fb_axis110_04Z(enIN_State       := enIN_State,
               parIN_Buttons    := ADR(AXIS.btTeachArAxis[Axis_e.ST110_04Z]),
               xIN_DisButtons   :=,
               xIN_Quit         := xIN_Quit,
               xIN_AX5000       := TRUE,
               xIN_ENC_ABS      := TRUE,
               xIN_PARAMok      := TRUE,
               xIN_FREE         := TRUE,
               xIN_FREE_HOME    := TRUE,
               rIN_POSMIN       := ST110_Axis.const110_04Z.POS_MIN,
               rIN_POSMAX       := ST110_Axis.const110_04Z.POS_MAX,
               rIN_VELOMAX      := ST110_Axis.const110_04Z.VELO_MAX,
               rIN_VELOMANU     := ST110_Axis.const110_04Z.VELO_MANU,
               rIN_VELOOPEN     := ST110_Axis.const110_04Z.VELO_MANU / 4,
               rIN_JogInc       := AXIS.rTeachIncAxis,
               rIN_VeloJogManu  := TO_REAL(AXIS.rJogVelo_pc),
               xIN_HomeExe      :=,
               xIN_HomeCalib    := FALSE,
               xIN_Execute      := fb_PnpVerAxisU.xOUT_Execute,
               xIN_Relative     := FALSE,
               rIN_Position     := LREAL_TO_REAL(fb_PnpVerAxisU.OUT_MoveProfile.lrPosition),
               rIN_Velocity     := LREAL_TO_REAL(fb_PnpVerAxisU.OUT_MoveProfile.lrVelocity),
               rIN_Acceleration := LREAL_TO_REAL(fb_PnpVerAxisU.OUT_MoveProfile.lrAccel),
               rIN_Deceleration := LREAL_TO_REAL(fb_PnpVerAxisU.OUT_MoveProfile.lrDecel),
               rIN_Jerk         := LREAL_TO_REAL(fb_PnpVerAxisU.OUT_MoveProfile.lrJerk),
               rIN_PosManu      :=
               TO_REAL(_20_AUTO.recipe
                           .linearAxis[LinearAxis_e.ST110_04Z].movesList[AXIS.bTeachPos[Axis_e.ST110_04Z]].lrPosition),
               xIN_Reset   := xIN_Reset,
               rOUT_ActPos => ST110_Axis.axis110_04Z.rActPos,
               axisIN_REF  := fb_simu_axis110_04Z.pOUT_axisRef^);

// pneumatics

fb_gripperLeft(xIN_Reset    := xIN_Reset OR (ST110_Pnp_e.RESET = iOUT_Step),
               xIN_Quit     := xIN_Quit,
               xIN_Manu     := enState.StateMANU = enIN_State,
               pbtIN_Button := ADR(HMI.btManuCylinders[StationList_e.ST110][1]),
               xIN_GS       := simu_gripperLeft.xOUT_inGS,
               xIN_AS       := simu_gripperLeft.xOUT_inAS,
               xIN_FREE     := TRUE,
               xINtoGS      := (ST110_Pnp_e.Vacum_off = iOUT_Step) OR (ST110_Pnp_e.Init_stop_vacum = iOUT_Step),
               xINtoAS      := _20_AUTO.recipe.st110.xUseVerLeft AND (ST110_Pnp_e.Vacum_on = iOUT_Step),
               tIN_ErrAS    := DINT_TO_TIME(_20_AUTO.recipe.cylinder2Pos[StationList_e.ST110]
                                                [ST110_Cylinders_e.VakuumgreiferLinks].toAS_alarm_time),
               tIN_ErrGS := DINT_TO_TIME(_20_AUTO.recipe.cylinder2Pos[StationList_e.ST110]
                                             [ST110_Cylinders_e.VakuumgreiferLinks].toGS_alarm_time),
               tIN_WaitAS := DINT_TO_TIME(_20_AUTO.recipe.cylinder2Pos[StationList_e.ST110]
                                              [ST110_Cylinders_e.VakuumgreiferLinks].toAS_wait_time),
               tIN_WaitGS := DINT_TO_TIME(_20_AUTO.recipe.cylinder2Pos[StationList_e.ST110]
                                              [ST110_Cylinders_e.VakuumgreiferLinks].toGS_wait_time));

simu_gripperLeft(xIN_Enable := TRUE, // PNP_SIMULATION AND CONST.USE_SIMULATION,
                 xIN_inGS   := (IO_BOX.I5500_ST110_vakumkontrolle_links / TO_INT(16#FFFF / 100)) <=
                               _20_AUTO.recipe.st110.vakum_left_pc,
                 xIN_inAS := (IO_BOX.I5500_ST110_vakumkontrolle_links / TO_INT(16#FFFF / 100)) >
                             _20_AUTO.recipe.st110.vakum_left_pc,
                 xIN_valve := fb_gripperLeft.xOUT_VALVE,
                 tIN_GS_ms := 200,  //ms
                 tIN_AS_ms := 200); //ms

fb_gripperRight(xIN_Reset    := xIN_Reset OR (ST110_Pnp_e.RESET = iOUT_Step),
                xIN_Quit     := xIN_Quit,
                xIN_Manu     := enState.StateMANU = enIN_State,
                pbtIN_Button := ADR(HMI.btManuCylinders[StationList_e.ST110][2]),
                xIN_GS       := simu_gripperRight.xOUT_inGS,
                xIN_AS       := simu_gripperRight.xOUT_inAS,
                xIN_FREE     := TRUE,
                xINtoGS      := (ST110_Pnp_e.Vacum_off = iOUT_Step) OR (ST110_Pnp_e.Init_stop_vacum = iOUT_Step),
                xINtoAS      := _20_AUTO.recipe.st110.xUseVerRight AND (ST110_Pnp_e.Vacum_on = iOUT_Step),
                tIN_ErrAS    := DINT_TO_TIME(_20_AUTO.recipe.cylinder2Pos[StationList_e.ST110]
                                                 [ST110_Cylinders_e.VakuumgreiferRechts].toAS_alarm_time),
                tIN_ErrGS := DINT_TO_TIME(_20_AUTO.recipe.cylinder2Pos[StationList_e.ST110]
                                              [ST110_Cylinders_e.VakuumgreiferRechts].toGS_alarm_time),
                tIN_WaitAS := DINT_TO_TIME(_20_AUTO.recipe.cylinder2Pos[StationList_e.ST110]
                                               [ST110_Cylinders_e.VakuumgreiferRechts].toAS_wait_time),
                tIN_WaitGS := DINT_TO_TIME(_20_AUTO.recipe.cylinder2Pos[StationList_e.ST110]
                                               [ST110_Cylinders_e.VakuumgreiferRechts].toGS_wait_time));

simu_gripperRight(xIN_Enable := TRUE, // PNP_SIMULATION AND CONST.USE_SIMULATION,
                  xIN_inGS   := (IO_BOX.I5600_ST110_vakumkontrolle_rechts / TO_INT(16#FFFF / 100)) <=
                                _20_AUTO.recipe.st110.vakum_right_pc,
                  xIN_inAS := (IO_BOX.I5600_ST110_vakumkontrolle_rechts / TO_INT(16#FFFF / 100)) >
                              _20_AUTO.recipe.st110.vakum_right_pc,
                  xIN_valve := fb_gripperRight.xOUT_VALVE,
                  tIN_GS_ms := 200,  //ms
                  tIN_AS_ms := 200); //ms

// kraft sensor
fb_kraftLeft(lrIN_MaxLimit := LREAL#2.0);
fb_kraftRight(lrIN_MaxLimit := LREAL#2.0);

(*******************************************************************)
(* OUTPUTS *)
(*******************************************************************)
// Error Flag 
xOUT_ErrFlag := (bOUT_Error <> 0) OR (ST110_Pnp_e.ERROR = iOUT_Step);
// Baustein befindet sich im Ablauf 
xOUT_Busy := (iOUT_Step > ST110_Pnp_e.READY) AND (iOUT_Step < ST110_Pnp_e.DONE);
// Baustein hat den Ablauf beendet
xOUT_Done := (iOUT_Step = ST110_Pnp_e.DONE);
// Process ready
xOUT_Ready := (iOUT_Step = ST110_Pnp_e.READY) OR (iOUT_Step = ST110_Pnp_e.waitOnMover);
// Timeout FB 				 		
xOUT_Timeout := TON_Timeout.Q;
// Itialisierung fertig			
xOUT_InitDone := (iOUT_Step = ST110_Pnp_e.READY) OR (iOUT_Step = ST110_Pnp_e.waitOnMover);
// Aktueller Schritt			
iOUT_Step := iOUT_Step; //Im Ablauf gesetzt		
sOUT_Step := TO_STRING(iOUT_Step);
//Fehlernummer	 
bOUT_Error := bOUT_Error; //Im Ablauf/FB gesetzt	
(* Warte (alle Schritte wo auf FG oder Teile gewartet wird) *)
xOUT_Wait := (iOUT_Step = ST110_Pnp_e.DONE) OR
             (iOUT_Step = ST110_Pnp_e.READY) OR
             (iOUT_Step = ST110_Pnp_e.START) OR
             (iOUT_Step = ST110_Pnp_e.waitOnMover) OR
             (iOUT_Step = ST110_Pnp_e.SYNC_MOVER_LEAVE) OR
             (iOUT_Step = ST110_Pnp_e.PnP_WaitOnFeeder);

xOUT_MoverFree := iOUT_Step >= ST110_Pnp_e.MOVER_FREE_OP AND iOUT_Step < ST110_Pnp_e.MOVER_NEEDED_OP;

iOUT_ProcessCompletion := F_GetPercent_2(iOUT_Step,
                                         ST110_Pnp_e.PnP_Hor_ToRotTablePos,
                                         ST110_Pnp_e.PnP_Hor_ToTrackPos,
                                         ST110_Pnp_e.PnP_Ver_ShuttleDown,
                                         ST110_Pnp_e.PnP_Ver_ShuttleUp);

xOUT_PickPiece := iOUT_Step = ST110_Pnp_e.PnP_Hor_ToTrackPos;

OUT.Q104_ST110_vacum_on_left  := fb_gripperLeft.xOUT_VALVE AND NOT (PNP_SIMULATION AND CONST.USE_SIMULATION);
OUT.Q105_ST110_vacum_on_right := fb_gripperRight.xOUT_VALVE AND NOT (PNP_SIMULATION AND CONST.USE_SIMULATION);

IF NOT IN.I004_druckwachter_luftdruck_ok THEN
    xIsPiecesPicked := FALSE;
END_IF

(*******************************************************************)
(* Ablauf *)
(*******************************************************************)

(* Sperren *)
IF xIN_Sperre THEN
    iPreStep  := ST110_Pnp_e.RESET;
    iOUT_Step := ST110_Pnp_e.RESET;
    RETURN;
END_IF;

(* Schritt Merker *)
IF iAktStep <> iOUT_Step THEN
    iLastStep := iAktStep;
    iAktStep  := iOUT_Step;
END_IF

(* START *)
rtSTART(CLK := xIN_Start);

IF 0 = bOUT_Error THEN
    IF fb_axis110_01Y.xOUT_ErrFlag THEN
        bOUT_Error := ST110_Alarm_e.Axis_110_01Y_error;
    ELSIF fb_axis110_02Z.xOUT_ErrFlag THEN
        bOUT_Error := ST110_Alarm_e.Axis_110_02Z_error;
    ELSIF fb_axis110_03Z.xOUT_ErrFlag THEN
        bOUT_Error := ST110_Alarm_e.Axis_110_03Z_error;
    ELSIF fb_axis110_04Z.xOUT_ErrFlag THEN
        bOUT_Error := ST110_Alarm_e.Axis_110_04Z_error;
    ELSIF fb_gripperLeft.xOUT_ErrFlag THEN
        bOUT_Error := ST110_Alarm_e.Cylinder_vacuum_griper_left;
    ELSIF fb_gripperRight.xOUT_ErrFlag THEN
        bOUT_Error := ST110_Alarm_e.Cylinder_vacuum_griper_right;
    END_IF
ELSIF iOUT_Step < ST110_Pnp_e.ERROR THEN
    iPreStep  := ST110_Pnp_e.INIT;
    iOUT_Step := ST110_Pnp_e.ERROR;
END_IF

(*******************************************************************)
(* Schrittkette  *)
(*******************************************************************)
CASE iOUT_Step OF

(***** RESET *****)
ST110_Pnp_e.RESET: (* Schritt 0-99 *)
    //Initialisierungen
    //Start Init Ablauf
    IF xIN_Init THEN
        iOUT_Step := ST110_Pnp_e.INIT;
        //Start Manu Ablauf
    ELSIF enIN_State = StateMANU AND xIN_NextStep THEN
        iOUT_Step := ST110_Pnp_e.INIT;
    END_IF;

(***** INIT *****)
ST110_Pnp_e.INIT: (* Grundstellung ? *)
    iOUT_Step := ST110_Pnp_e.Init_VerticalUp_04;

ST110_Pnp_e.Init_VerticalUp_04:
    IF fb_PnpVerAxisU.MoveTo(ST110_PnpVerPushPos_e.down).xOUT_InPos THEN
        iOUT_Step := ST110_Pnp_e.Init_VerticalUp_02_03;

    END_IF

ST110_Pnp_e.Init_VerticalUp_02_03:
    IF fb_gripperLeft.xIN_AS OR fb_gripperRight.xIN_AS THEN
        IF fb_PnpVerAxisL.MoveTo(ST110_PnpVerPos_e.UpFull).xOUT_InPos AND
           fb_PnpVerAxisR.MoveTo(ST110_PnpVerPos_e.UpFull).xOUT_InPos THEN
            IF fb_axis110_01Y.xOUT_READY OR fb_axis110_01Y.xOUT_HOMED THEN
                iOUT_Step := ST110_Pnp_e.Init_HorizontalsToTrack;
            ELSE
                iOUT_Step := ST110_Pnp_e.Init_HomeHorizontals;
            END_IF
        END_IF
    ELSE
        IF fb_PnpVerAxisL.MoveTo(ST110_PnpVerPos_e.UpEmpty).xOUT_InPos AND
           fb_PnpVerAxisR.MoveTo(ST110_PnpVerPos_e.UpEmpty).xOUT_InPos THEN
            IF fb_axis110_01Y.xOUT_READY OR fb_axis110_01Y.xOUT_HOMED THEN
                iOUT_Step := ST110_Pnp_e.Init_HorizontalsToTrack;
            ELSE
                iOUT_Step := ST110_Pnp_e.Init_HomeHorizontals;
            END_IF
        END_IF
    END_IF

ST110_Pnp_e.Init_HomeHorizontals:
    fb_axis110_01Y.rIN_Velocity :=
        _20_AUTO.recipe.linearAxis[LinearAxis_e.ST110_01Y].movesList[ST110_PnpHorPos_e.GS].lrVelocity;

    IF fb_axis110_01Y.xOUT_HOMED THEN
        iOUT_Step := ST110_Pnp_e.Init_HorizontalsToTrack;
    END_IF

ST110_Pnp_e.Init_HorizontalsToTrack:
    IF fb_PnpHorAxis.MoveTo(ST110_PnpHorPos_e.GS).xOUT_InPos THEN
        IF NOT xIsPiecesPicked THEN
            iOUT_Step := ST110_Pnp_e.Init_stop_vacum;
        ELSE
            iOUT_Step := ST110_Pnp_e.Init_check_if_pces_handled;
        END_IF
    END_IF

ST110_Pnp_e.Init_stop_vacum:
    iOUT_Step := ST110_Pnp_e.Init_check_if_pces_handled;

ST110_Pnp_e.Init_check_if_pces_handled:
    IF (NOT _20_AUTO.recipe.st110.xUseVerLeft AND fb_gripperLeft.xOUT_inAS) OR
       (NOT _20_AUTO.recipe.st110.xUseVerRight AND fb_gripperRight.xOUT_inAS) THEN
        // ERROR: a piece is present in an unused gripper
        bOUT_Error := ST110_Alarm_e.Piece_in_unused_griper;
        iOUT_Step  := ST110_Pnp_e.ERROR;

    ELSIF _20_AUTO.recipe.st110.xUseVerLeft AND
          NOT fb_gripperLeft.xOUT_inAS AND
          _20_AUTO.recipe.st110.xUseVerRight AND
          fb_gripperRight.xOUT_inAS THEN
        // ERROR:  Initialisation failed. A piece is missing in the left griper.
        bOUT_Error := ST110_Alarm_e.Piece_missing_left_griper;
        iOUT_Step  := ST110_Pnp_e.ERROR;

    ELSIF _20_AUTO.recipe.st110.xUseVerLeft AND
          fb_gripperLeft.xOUT_inAS AND
          _20_AUTO.recipe.st110.xUseVerRight AND
          NOT fb_gripperRight.xOUT_inAS THEN
        // ERROR:  Initialisation failed. A piece is missing in the right griper.
        bOUT_Error := ST110_Alarm_e.Piece_missing_right_griper;
        iOUT_Step  := ST110_Pnp_e.ERROR;

    ELSIF (NOT fb_gripperLeft.xOUT_inAS AND NOT fb_gripperRight.xOUT_inAS) OR NOT xIsPiecesPicked THEN
        iOUT_Step := ST110_Pnp_e.READY;

    ELSE
        iOUT_Step := ST110_Pnp_e.waitOnMover;
    END_IF

(***** READY / INIT DONE *****)
ST110_Pnp_e.READY:    (* Start AUTO,END,LEER,STEP *)
    IF xIN_Start THEN //IF rtSTART.Q THEN
        iOUT_Step := ST110_Pnp_e.START;
    END_IF

(***** START  ZYKLISCH *****)
ST110_Pnp_e.START: (*  *)
    IF xIN_NextStep AND pxFG_Freigabe^ THEN
        IF enState.StateLEER = enIN_State THEN
            IF __ISVALIDREF(Mover) THEN
                IF Mover.GetLastStationDone() > 0 THEN
                    iOUT_Step := ST110_Pnp_e.PnP_Hor_ToRotTablePos;
                ELSE
                    iOUT_Step := ST110_Pnp_e.waitOnMover;
                END_IF
            END_IF
        ELSE
            iOUT_Step := ST110_Pnp_e.PnP_Hor_ToRotTablePos;
        END_IF
    END_IF;

ST110_Pnp_e.PnP_Hor_ToRotTablePos:
    IF xIN_NextStep AND fb_PnpHorAxis.MoveTo(ST110_PnpHorPos_e.AS).xOUT_InPos THEN
        iOUT_Step := ST110_Pnp_e.PnP_WaitOnFeeder;
    END_IF

ST110_Pnp_e.PnP_WaitOnFeeder:
    IF xIN_PceReadyToPick THEN
        iOUT_Step := ST110_Pnp_e.PnP_Ver_RotTableDown;
    END_IF

ST110_Pnp_e.PnP_Ver_RotTableDown:
    IF xIN_NextStep AND
       (fb_PnpVerAxisL.MoveTo(ST110_PnpVerPos_e.DownEmpty).xOUT_InPos OR
       NOT _20_AUTO.recipe.st110.xUseVerLeft) AND
       (fb_PnpVerAxisR.MoveTo(ST110_PnpVerPos_e.DownEmpty).xOUT_InPos OR
       NOT _20_AUTO.recipe.st110.xUseVerRight) THEN
        iOUT_Step := ST110_Pnp_e.Vacum_on;
    END_IF;

ST110_Pnp_e.Vacum_on:
    IF xIN_NextStep AND
       (NOT _20_AUTO.recipe.st110.xUseVerLeft OR simu_gripperLeft.xOUT_inAS) AND
       (NOT _20_AUTO.recipe.st110.xUseVerRight OR simu_gripperRight.xOUT_inAS) THEN
        iOUT_Step       := ST110_Pnp_e.PnP_Ver_RotTableUp;
        xIsPiecesPicked := TRUE;
    END_IF;

ST110_Pnp_e.PnP_Ver_RotTableUp:
    IF xIN_NextStep AND
       (fb_PnpVerAxisL.MoveTo(ST110_PnpVerPos_e.UpFull).xOUT_InPos OR
       NOT _20_AUTO.recipe.st110.xUseVerLeft) AND
       (
       fb_PnpVerAxisR.MoveTo(ST110_PnpVerPos_e.UpFull).xOUT_InPos OR
       NOT _20_AUTO.recipe.st110.xUseVerRight
           ) THEN
        iOUT_Step := ST110_Pnp_e.PnP_Hor_ToTrackPos;
    END_IF;

ST110_Pnp_e.PnP_Hor_ToTrackPos:
    IF xIN_NextStep AND fb_PnpHorAxis.MoveTo(ST110_PnpHorPos_e.GS).xOUT_InPos THEN
        iOUT_Step := ST110_Pnp_e.waitOnMover;
    END_IF

ST110_Pnp_e.waitOnMover: (*  *)
    IF xIN_NextStep AND (__ISVALIDREF(Mover) OR HMI.bArForceCyclusState[StationList_e.ST110]) THEN
        IF Mover.GetLastStationDone() >= INT#110 THEN
            iOUT_Step := ST110_Pnp_e.SYNC_MOVER_LEAVE;
        ELSIF Mover.GetLastStationDone() < INT#105 THEN
            iOUT_Step := ST110_Pnp_e.SYNC_MOVER_LEAVE;
        ELSE
            iOUT_Step := ST110_Pnp_e.Pnp_Handling_pin_up;
        END_IF
    END_IF;

ST110_Pnp_e.Pnp_Handling_pin_up:
    IF xIN_NextStep AND fb_PnpVerAxisU.MoveTo(ST110_PnpVerPushPos_e.up).xOUT_InPos THEN
        iOUT_Step := ST110_Pnp_e.PnP_Ver_ShuttleDown;
    END_IF

ST110_Pnp_e.PnP_Ver_ShuttleDown:
    IF _20_AUTO.recipe.st110.xUseVerLeft THEN
        fb_PnpVerAxisL.MoveTo(ST110_PnpVerPos_e.DownFullQuick);
    END_IF

    IF _20_AUTO.recipe.st110.xUseVerRight THEN
        fb_PnpVerAxisR.MoveTo(ST110_PnpVerPos_e.DownFullQuick);
    END_IF

    IF xIN_NextStep AND
       (NOT _20_AUTO.recipe.st110.xUseVerLeft OR fb_axis110_02Z.xOUT_DONE) AND
       (NOT _20_AUTO.recipe.st110.xUseVerRight OR fb_axis110_03Z.xOUT_DONE) THEN
        iOUT_Step       := ST110_Pnp_e.PnP_Ver_StartTorqueControl;
        xIsPiecesPicked := FALSE;

        IF __ISVALIDREF(Mover) THEN
            IF NOT Mover.SetLastStation(110) THEN
                ASSERT(0);
            END_IF
        END_IF
    END_IF;

ST110_Pnp_e.PnP_Ver_StartTorqueControl:

    IF _20_AUTO.recipe.st110.xUseVerLeft AND NOT fb_axis110_02Z.xOUT_BUSY THEN
        fb_PnpVerAxisL.MoveTo(ST110_PnpVerPos_e.DownFullTorqueControl);
    END_IF

    IF _20_AUTO.recipe.st110.xUseVerRight AND NOT fb_axis110_03Z.xOUT_BUSY THEN
        fb_PnpVerAxisR.MoveTo(ST110_PnpVerPos_e.DownFullTorqueControl);
    END_IF

    IF (fb_axis110_02Z.xOUT_BUSY OR NOT _20_AUTO.recipe.st110.xUseVerLeft) AND
       (fb_axis110_03Z.xOUT_BUSY OR NOT _20_AUTO.recipe.st110.xUseVerRight) THEN
        iOUT_Step := ST110_Pnp_e.PnP_Ver_ShuttleTorqueControl;

    ELSIF (fb_PnpVerAxisL.xOUT_InPos OR NOT _20_AUTO.recipe.st110.xUseVerLeft) AND
          (fb_PnpVerAxisR.xOUT_InPos OR NOT _20_AUTO.recipe.st110.xUseVerRight) THEN
        bOUT_Error := ST110_Alarm_e.Reach_end_pos_without_needed_torque;

    END_IF

// We need a fb that enables for us torque control. Here we just go a bit further
ST110_Pnp_e.PnP_Ver_ShuttleTorqueControl:
    // If one of the axis have not started its movement, we do it again
    IF NOT fb_axis110_02Z.xOUT_BUSY AND NOT fb_axis110_03Z.xOUT_BUSY THEN
        iOUT_Step := ST110_Pnp_e.PnP_Ver_StartTorqueControl;
    END_IF

    IF (fb_PnpVerAxisL.xOUT_InPos OR NOT _20_AUTO.recipe.st110.xUseVerLeft) AND
       (fb_PnpVerAxisR.xOUT_InPos OR NOT _20_AUTO.recipe.st110.xUseVerRight) THEN
        IF (PNP_SIMULATION AND CONST.USE_SIMULATION) OR PNP_DONT_CHECK_KRAFT THEN
            iOUT_Step := ST110_Pnp_e.PnP_Ver_quick_stop;
        ELSE
            iOUT_Step := ST110_Pnp_e.ERROR;

        END_IF

    ELSIF
        (NOT _20_AUTO.recipe.st110.xUseVerLeft OR (fb_kraftLeft.lrOUT_value >= _20_AUTO.recipe.st110.kraft_left_raw)
            ) AND
        (NOT _20_AUTO.recipe.st110.xUseVerRight OR (fb_kraftRight.lrOUT_value >= _20_AUTO.recipe.st110.kraft_right_raw)
            ) THEN
        iOUT_Step := ST110_Pnp_e.PnP_Ver_quick_stop;
    END_IF;

ST110_Pnp_e.PnP_Ver_quick_stop:
    IF xIN_NextStep THEN
        iOUT_Step := ST110_Pnp_e.Vacum_off;
    END_IF;

ST110_Pnp_e.Vacum_off:
    IF xIN_NextStep AND fb_gripperLeft.xOUT_inGS AND fb_gripperRight.xOUT_inGS THEN
        iOUT_Step := ST110_Pnp_e.PnP_Ver_ShuttleUp;
    END_IF;

ST110_Pnp_e.PnP_Ver_ShuttleUp:
    IF xIN_NextStep AND
       (fb_PnpVerAxisL.MoveTo(ST110_PnpVerPos_e.UpEmpty).xOUT_InPos OR
       NOT _20_AUTO.recipe.st110.xUseVerLeft) AND
       (fb_PnpVerAxisR.MoveTo(ST110_PnpVerPos_e.UpEmpty).xOUT_InPos OR
       NOT _20_AUTO.recipe.st110.xUseVerRight) AND
       fb_PnpVerAxisU.MoveTo(ST110_PnpVerPushPos_e.down).xOUT_InPos THEN
        iOUT_Step := ST110_Pnp_e.SYNC_MOVER_LEAVE;

        IF __ISVALIDREF(Mover) THEN
            IF NOT Mover.SetLastStation(110) THEN
                ASSERT(0);
            END_IF
        END_IF
    END_IF;

ST110_Pnp_e.SYNC_MOVER_LEAVE:
    // The mover needs to be taken by MoverMan
    IF NOT __ISVALIDREF(Mover) THEN
        IF fb_gripperLeft.xOUT_inGS AND fb_gripperRight.xOUT_inGS THEN
            iOUT_Step := ST110_Pnp_e.DONE;
        ELSE
            iOUT_Step := ST110_Pnp_e.waitOnMover;
        END_IF
    END_IF

(***** DONE *****)
ST110_Pnp_e.DONE: (* Letzter Schritt  *)
    IF NOT xIN_AlarmAktiv THEN
        //AUTO
        IF (enIN_State = StateAUTO) AND xIN_RestartCYCL THEN
            iOUT_Step := ST110_Pnp_e.START;
            //STEP / END / LEERFAHREN restart
        ELSIF (enIN_State < StateAUTO) AND (enIN_State >= enState.StateSTEP) AND xIN_RestartCYCL THEN
            iOUT_Step := ST110_Pnp_e.START;
            //STEP / END / LEERFAHREN fertig
        ELSIF (enIN_State = StateREADY) THEN
            iOUT_Step := ST110_Pnp_e.READY;
        END_IF;
    END_IF;

(************ ERROR *************)
ST110_Pnp_e.ERROR: (* ERROR *) ;

END_CASE;

END_FUNCTION_BLOCK

// ---- POUs/20_AUTO/Simu/FB_Simu_AxisLIN_V1_1.TcPOU
FUNCTION_BLOCK FB_Simu_AxisLIN_V1_1
VAR_INPUT
    xIN_InSimu    : BOOL;
    rIN_PosActual : REAL;

    pIN_axisSimu : POINTER TO AXIS_REF; // simulation axis ref, without hardware connection
    pIN_axisHW   : POINTER TO AXIS_REF; // hardware axis ref, the one wich is connected to hardware

    rIN_PosMax : REAL;
    rIN_PosMin : REAL;
    rIN_PixMax : INT;
    rIN_PixMin : INT;
END_VAR
VAR_OUTPUT
    rOUT_PixActual : INT;                 // actual relative position of the axis
    pOUT_axisRef   : POINTER TO AXIS_REF; // current axis ref used
END_VAR
VAR
	power_real_axis : MC_Power;
	reset_real_axis : MC_Reset;
END_VAR

VAR_IN_OUT
    //xIN_InSimu    : BOOL;
END_VAR

rOUT_PixActual := MAP_REAL_TO_INT(rValue    := rIN_PosActual,
                                  rFromHigh := rIN_PosMax,
                                  rFromLow  := rIN_PosMin,
                                  rToHigh   := rIN_PixMax,
                                  rToLow    := rIN_PixMin);

IF xIN_InSimu THEN
    pOUT_axisRef := pIN_axisSimu;
    power_real_axis(Axis            := pIN_axisHW^,
                    Enable          := NOT power_real_axis.Error,
                    Enable_Positive := TRUE,
                    Enable_Negative := TRUE);

    reset_real_axis(Axis    := pIN_axisHW^,
                    Execute := power_real_axis.Error);
ELSE
    pOUT_axisRef := pIN_axisHW;
END_IF

END_FUNCTION_BLOCK

// ---- POUs/20_AUTO/ST110/FB_ABL_110_Feeder.TcPOU
FUNCTION_BLOCK FB_ABL_110_Feeder
(****************************************************************************************)
(*	TITEL				RFID-Ring laden, Feeder and rotary table                        *)
(*	Status				ungetestet                         								*)
(*	Beschrieb:			Ablaufbeschreibung												*)
(*																						*)
(*	Steps:	self-explained using enum													*)
(***********************************Revisionen*******************************************)
(*	see github blames																	*)
(****************************************************************************************)

VAR_INPUT
    xIN_Reset       : BOOL;          // Schrittkette zurücksetzen 
    xIN_Init        : BOOL;          // Initialisieren
    xIN_Quit        : BOOL;          // Fehler quittieren 
    xIN_Start       : BOOL;          // Startbefehl
    xIN_Sperre      : BOOL;          // FB Sperren 
    xIN_NextStep    : BOOL;          // Nächsten Schritt ausführen 
    xIN_AlarmAktiv  : BOOL;          // Anlage hat Alarm
    xIN_DryCycle    : BOOL;          // Fahren ohne Teile
    xIN_RestartCYCL : BOOL;          // Zyklus erneut starten im STEP, END, LEERFAHREN
    enIN_State      : enState;       // Status Anlage
    tIN_Timeout     : TIME := T#10s; // Timout

    pxFG_Freigabe : POINTER TO BOOL; //Freigabe von Station

    // Application specific
    xIN_PickPiece : BOOL; (* signal from the pick and place element
                             the number of picked signal depend on the recipe *)
    xIN_RotTableBlockedByPnp : BOOL; // Is the pick and place blocking the rotary table?
END_VAR
VAR_OUTPUT
    (* standart Ausgänge *)
    xOUT_ErrFlag  : BOOL;           // Error Flag 
    xOUT_Busy     : BOOL;           // Baustein befindet sich im Ablauf 
    xOUT_Done     : BOOL;           // Baustein hat den Ablauf beendet 		
    xOUT_Ready    : BOOL;           // Ready to begin, should be the same state as done	
    xOUT_Timeout  : BOOL;           // Timeout FB 
    xOUT_InitDone : BOOL;           // initialisierung fertig
    xOUT_Wait     : BOOL;           // Wartet auf Bedingung
    iOUT_Step     : ST110_Feeder_e; // Aktueller Schritt 
    sOUT_Step     : STRING;         // Aktueller Schritt but in string format
    bOUT_Error    : BYTE;           // Fehlernummer

    // Application specific
    xOUT_PceReadyToPick : BOOL; // the piece(s) is/are ready to picked
END_VAR
VAR
    (* Standard *)
    (* Schritt *)
    iLastStep : ST110_Feeder_e; // Merker letzter Schritt 
    iPreStep  : ST110_Feeder_e; // Schritt zurück nach Alarm 
    iAktStep  : ST110_Feeder_e; // aktueller Schritt

    // Trigger Starten 
    rtSTART : R_TRIG;
    // Timer TimeOut 
    TON_Timeout : TON;

    (* Bausteine *)
	btfb_feeder					: FB_BUTTON;

    // Application specific
    fb_axis110_10W               : FB_AxisLMturn_V1_1;
    simu_axis110_10W             : FB_Simu_AxisLM_V1_1;
    fb_feeder                    : FB_Feeder2Sensors;
    fifo                         : FB_Fifo(3);
    simu_feeder                  : FB_Simu_Feeder; // simulation of a feeder
    simu_fifo_feeder_to_rotTable : FB_Fifo(20);    // fifo to hold a piece
    rtPutPiece                   : R_TRIG;         // trigger to add a piece

    rtPick : R_TRIG; // r_trig signal from the pick and place machine

    iCurrentTableIndex : INT; // current table index
    iSearchIndex       : INT; (* Initialization index TO see how many element we have AT startup
                                 or after an alarm *)

    ton_wait_blow_piece : TON;
    tof_color_sensor    : TOF;

	rTest : REAL;
END_VAR
VAR CONSTANT
    MAX_SEARCH_TURN : INT := 3; // maximum search number

    FEEDER_SIMULATION : BOOL := FALSE; // Simulate this code
END_VAR

(*******************************************************************)
(* Trigger  *)
(*******************************************************************)
(* Zurücksetzen *)
IF xIN_RESET THEN
    iPreStep  := ST110_Feeder_e.RESET;
    iOUT_Step := ST110_Feeder_e.RESET;
END_IF;

(* Error Quittieren *)
IF (bOUT_Error <> 0) AND xIN_Quit THEN
    xOUT_ErrFlag := FALSE;
    bOUT_Error   := 0;
    iOUT_Step    := iPreStep;
END_IF;

iCurrentTableIndex := iCurrentTableIndex MOD 3;

(*******************************************************************)
(* Timer *)
(*******************************************************************)
TON_Timeout(IN := xIN_NextStep AND (iLastStep = iOUT_Step) (*todo FG *) ,
            PT := tIN_Timeout);

// we use a set reset to be sure that the blower blow event if the time
// is not elapsed
IF IO_BOX.I8004_ST110_farbsensor_lagekontrolle THEN
    ton_wait_blow_piece.IN := TRUE;

ELSIF NOT IO_BOX.I8004_ST110_farbsensor_lagekontrolle AND ton_wait_blow_piece.Q THEN
    ton_wait_blow_piece.IN := FALSE;

END_IF

ton_wait_blow_piece(IN :=, // see code above
                    PT := DINT_TO_TIME(_20_AUTO.recipe.st110.waitBlowPieceTon_ms));

tof_color_sensor(IN := ton_wait_blow_piece.Q,
                 PT := DINT_TO_TIME(_20_AUTO.recipe.st110.blowPieceTof_ms));

(*******************************************************************)
(* Bausteine *)
(*******************************************************************)
btfb_feeder(pbtIN  := ADR(HMI.btManuCylinders[StationList_e.ST110][3]),
            xINdis := (enIN_State <> enState.StateMANU),
            xINon  :=,
            xINerr := fb_feeder.xOUT_Empty);

IF btfb_feeder.pbtIN^.rtrig THEN
    btfb_feeder.xINon := NOT btfb_feeder.xINon;
ELSIF (enIN_State <> enState.StateMANU) THEN
    btfb_feeder.xINon := FALSE;
END_IF;

fb_feeder(xIN_Enable                := (enIN_State > enState.StateEND) OR btfb_feeder.xINon,
          xIN_PieceInEnd            := IO_BOX.I8001_ST110_maximum,
          xIN_PieceMax              := IO_BOX.I8001_ST110_maximum,
          xIN_InSimulation          := FEEDER_SIMULATION AND CONST.USE_SIMULATION,
          refIN_SimulatedFifo       := simu_fifo_feeder_to_rotTable,
          iIN_FifoSetMaxSensorValue := 10,
          diIN_SignlFilter_ms       := _20_AUTO.recipe.st110.FeederConfig.InFilterDelay,
          diIN_StartDelay_ms        := _20_AUTO.recipe.st110.FeederConfig.StartDelay,
          diIN_StopDelay_ms         := _20_AUTO.recipe.st110.FeederConfig.StopDelay,
          diIN_EmptyDelay_ms        := _20_AUTO.recipe.st110.FeederConfig.EmptyDelay);

simu_feeder(xIN_Enable         := fb_feeder.xOUT_EnableFeeder AND FEEDER_SIMULATION AND CONST.USE_SIMULATION,
            xIN_PceSensor      := fb_feeder.xIN_PieceInEnd,
            tIN_NewPieceTime   := 500,
            iIN_WaitTimeMin_ms := 500,
            iIN_WaitTimeMax_ms := 1000);

rtPick(CLK := xIN_PickPiece);
rtPutPiece(CLK := simu_feeder.xOUT_NewPiece);

IF rtPutPiece.Q AND NOT simu_fifo_feeder_to_rotTable.IsFull() THEN
    simu_fifo_feeder_to_rotTable.Put(1);
END_IF

IF ST110_Feeder_e.Init_simu_home_table = iOUT_Step THEN
    fb_axis110_10W.rIN_Position := TO_REAL(120.0 - LMOD(ST110_Axis.axis110_10W.rActPos, 120.0));

ELSE
    fb_axis110_10W.rIN_Position := 120.0;

END_IF

simu_axis110_10W(xIN_Enable          := FEEDER_SIMULATION AND CONST.USE_SIMULATION,
                 wIN_AxisState       := ST110_Axis.axis110_10W.wState,
                 bIN_AxisCntr        := fb_axis110_10W.bOUT_AxisCntr,
                 udiIN_HomingTime_ms := 1000,
                 pIN_axisSimu        := ADR(SIMU.axis_ref[Axis_e.ST110_10W]),
                 pIN_axisHW          := ADR(ST110_Axis.axis110_10W.axis),
                 rIN_PosActual       := fb_axis110_10W.rOUT_ActPos,
                 rIN_PosMax          := ST110_Axis.const110_10W.POS_MAX,
                 rIN_PosMin          := ST110_Axis.const110_10W.POS_MIN,
                 rIN_PixMax          := 0,
                 rIN_PixMin          := 0);

fb_axis110_10W(enIN_State     := enIN_State,
               parIN_Buttons  := ADR(AXIS.btTeachArAxis[Axis_e.ST110_10W]),
               xIN_DisButtons :=,
               xIN_Quit       := xIN_Quit,
               xIN_PARAMok    := TRUE,
               xIN_FREE       := NOT xIN_RotTableBlockedByPnp,
               xIN_FREE_HOME  := TRUE,
               rIN_POSMIN     := ST110_Axis.const110_10W.POS_MIN,
               rIN_POSMAX     := ST110_Axis.const110_10W.POS_MAX,
               rIN_VELOMAX    := ST110_Axis.const110_10W.VELO_MAX,
               rIN_VELOMANU   := ST110_Axis.const110_10W.VELO_MANU,
               rIN_VELOOPEN   := ST110_Axis.const110_10W.VELO_MANU / 4,
               rIN_JogInc     := AXIS.rTeachIncAxis,
               xIN_Execute    := ST110_Feeder_e.Init_set_table_pos = iOUT_Step OR
                                 ST110_Feeder_e.Init_table_go_to_zero = iOUT_Step OR
                                 ST110_Feeder_e.Init_simu_home_table = iOUT_Step OR
                                 ST110_Feeder_e.load_piece = iOUT_Step OR
                                 ST110_Feeder_e.wait_rotary_table_done = iOUT_Step,
               xIN_Relative     := fb_axis110_10W.xIN_Execute,
               xIN_STOP         := FALSE,
               xIN_OFF          := FALSE,
               rIN_Position     :=, // Is set above
               rIN_Velocity     := TO_REAL(100.0),
               rIN_Acceleration := TO_REAL(1440.0),
               rIN_Deceleration := TO_REAL(1440.0),
               rIN_Jerk         := TO_REAL(720000.0),
               xIN_Home         := ST110_feeder_e.Init_home_table = iOUT_Step,
               xIN_Reset        := xIN_Reset OR ST110_feeder_e.RESET = iOUT_Step,
               // The simu fb gives us the hardware signal when we are not in simulation
               wAxisState    := simu_axis110_10W.wOUT_AxisState,
               bOUT_AxisCntr => ST110_Axis.axis110_10W.bCtrlHi,
               rOUT_ActPos   =>, // leave empty, rActPos must be set using the modulo
               axisIN_REF    := simu_axis110_10W.pOUT_axisRef^);

ST110_Axis.axis110_10W.rActPos := LREAL_TO_REAL(simu_axis110_10W.pOUT_axisRef^.NcToPlc.ModuloActPos);

(*******************************************************************)
(* OUTPUTS *)
(*******************************************************************)
// Error Flag 
xOUT_ErrFlag := (bOUT_Error <> 0) OR (ST110_Feeder_e.ERROR = iOUT_Step);
// Baustein befindet sich im Ablauf 
xOUT_Busy := (iOUT_Step > ST110_Feeder_e.READY) AND (iOUT_Step < ST110_Feeder_e.DONE);
// Baustein hat den Ablauf beendet
xOUT_Done := (iOUT_Step = ST110_Feeder_e.DONE);
// Process ready
xOUT_Ready := (iOUT_Step = ST110_Feeder_e.READY);
// Timeout FB 				 		
xOUT_Timeout := TON_Timeout.Q;
// Itialisierung fertig			
xOUT_InitDone := (iOUT_Step = ST110_Feeder_e.READY);
// Aktueller Schritt			
iOUT_Step := iOUT_Step; //Im Ablauf gesetzt		
sOUT_Step := TO_STRING(iOUT_Step);
//Fehlernummer	 
bOUT_Error := bOUT_Error; //Im Ablauf/FB gesetzt	
(* Warte (alle Schritte wo auf FG oder Teile gewartet wird) *)
xOUT_Wait := (iOUT_Step = ST110_Feeder_e.DONE) OR
             (iOUT_Step = ST110_Feeder_e.READY);

// TODO add simulation constant to prevent the output to be set
IO_BOX.Q8000_ST110_freigabe_wf    := fb_feeder.xOUT_EnableFeeder AND NOT (FEEDER_SIMULATION AND CONST.USE_SIMULATION);
IO_BOX.Q8003_ST110_forderband_ein :=
    (enIN_State >= enState.StateLEER) AND
    NOT (FEEDER_SIMULATION AND CONST.USE_SIMULATION);

// blow out

IO_BOX.Q8005_ST110_blow_piece := fb_feeder.xOUT_EnableFeeder AND
                                 tof_color_sensor.Q AND
                                 NOT (FEEDER_SIMULATION AND CONST.USE_SIMULATION);

(*******************************************************************)
(* Ablauf *)
(*******************************************************************)

(* Sperren *)
IF xIN_Sperre THEN
    iPreStep  := ST110_Feeder_e.RESET;
    iOUT_Step := ST110_Feeder_e.RESET;
    RETURN;
END_IF;

(* Schritt Merker *)
IF iAktStep <> iOUT_Step THEN
    iLastStep := iAktStep;
    iAktStep  := iOUT_Step;
END_IF

(* START *)
rtSTART(CLK := xIN_Start);

IF 0 = bOUT_Error THEN
    IF fb_axis110_10W.xOUT_ErrFlag THEN
        bOUT_Error := ST110_Alarm_e.Axis_110_10W_error;
		
	ELSIF NOT IO_BOX.I8002_ST110_alarm_forderband THEN
        bOUT_Error := ST110_Alarm_e.Feeder_error;
	
    END_IF
ELSIF iOUT_Step < ST110_Feeder_e.ERROR THEN
    iOUT_Step := ST110_Feeder_e.ERROR;
END_IF

(*******************************************************************)
(* Schrittkette  *)
(*******************************************************************)
CASE iOUT_Step OF

(***** RESET *****)
ST110_Feeder_e.RESET: (* Schritt 0-99 *)
    //Initialisierungen
    //Start Init Ablauf
    IF xIN_Init THEN
        iOUT_Step := ST110_Feeder_e.INIT;
        //Start Manu Ablauf
    ELSIF enIN_State = StateMANU AND xIN_NextStep THEN
        iOUT_Step := ST110_Feeder_e.INIT;
    END_IF;

(***** INIT *****)
ST110_Feeder_e.INIT: (* Grundstellung ? *)
    IF NOT xIN_RotTableBlockedByPnp THEN
        iOUT_Step := ST110_Feeder_e.Init_home_table;
    END_IF

ST110_Feeder_e.Init_home_table:
    IF fb_axis110_10W.xOUT_HOMED THEN
        iCurrentTableIndex := 0;

        IF FEEDER_SIMULATION AND CONST.USE_SIMULATION THEN
            iOUT_Step := ST110_Feeder_e.Init_simu_home_table;
        ELSE
            iOUT_Step := ST110_Feeder_e.Init_reset_search_index;
        END_IF
    END_IF

ST110_Feeder_e.Init_simu_home_table:
    IF fb_axis110_10W.xOUT_DONE THEN
        iOUT_Step := ST110_Feeder_e.Init_reset_search_index;
    END_IF

ST110_Feeder_e.Init_table_go_to_zero:
    IF fb_axis110_10W.xOUT_DONE THEN
        iOUT_Step := ST110_Feeder_e.Init_reset_search_index;
    END_IF

ST110_Feeder_e.Init_reset_search_index:
    iSearchIndex := 0;
    fifo.Empty();
    iOUT_Step := ST110_Feeder_e.READY; // Bypass search algorithm, unusful

ST110_Feeder_e.Init_set_table_pos:
    IF fb_axis110_10W.xOUT_DONE THEN
        iCurrentTableIndex := iCurrentTableIndex + 1;
        iOUT_Step          := ST110_Feeder_e.Init_see_if_piece_there;
    END_IF

ST110_Feeder_e.Init_see_if_piece_there:
    IF simu_feeder.xOUT_NewPiece THEN
        fifo.Put(1);
    END_IF

    IF iSearchIndex < MAX_SEARCH_TURN THEN
        iOUT_Step    := ST110_Feeder_e.Init_set_table_pos;
        iSearchIndex := iSearchIndex + 1;
    ELSE
        iOUT_Step := ST110_Feeder_e.READY;
    END_IF

(***** READY / INIT DONE *****)
ST110_Feeder_e.READY: (* Start AUTO,END,LEER,STEP *)
    IF xIN_Start THEN //IF rtSTART.Q THEN
        iOUT_Step := ST110_Feeder_e.START;
    END_IF

(***** START  ZYKLISCH *****)
ST110_Feeder_e.START: (*  *)
    IF xIN_NextStep AND pxFG_Freigabe^ THEN
        iOUT_Step := ST110_Feeder_e.check_if_feeding_necessary;
    END_IF;

ST110_Feeder_e.check_if_feeding_necessary:
    IF fifo.IsFull() THEN
        iOUT_Step := ST110_Feeder_e.DONE;
    ELSE
        iOUT_Step := ST110_Feeder_e.wait_on_a_piece;
    END_IF

ST110_Feeder_e.wait_on_a_piece:
    IF (FEEDER_SIMULATION AND CONST.USE_SIMULATION AND NOT simu_fifo_feeder_to_rotTable.IsEmpty()) OR
       (NOT (FEEDER_SIMULATION AND CONST.USE_SIMULATION) AND IO_BOX.I6000_ST110_teil_in_vereinzelung) THEN
        iOUT_Step := ST110_Feeder_e.load_piece;
        simu_fifo_feeder_to_rotTable.Pop(1);
    END_IF

ST110_Feeder_e.load_piece:
    IF NOT fb_axis110_10W.xOUT_DONE THEN
        iOUT_Step := ST110_Feeder_e.wait_rotary_table_done;
    END_IF

ST110_Feeder_e.wait_rotary_table_done:
    IF fb_axis110_10W.xOUT_DONE THEN
        fifo.Put(1);
        iOUT_Step := ST110_Feeder_e.check_if_feeding_necessary;
    END_IF

(***** DONE *****)
ST110_Feeder_e.DONE: (* Letzter Schritt  *)
    IF rtPick.Q THEN
        fifo.Pop(TO_INT(_20_AUTO.recipe.st110.xUseVerLeft));
        fifo.Pop(TO_INT(_20_AUTO.recipe.st110.xUseVerRight));
    END_IF

    IF NOT xIN_AlarmAktiv THEN
        //AUTO
        IF (enIN_State = StateAUTO) AND xIN_RestartCYCL AND NOT fifo.IsFull() THEN
            iOUT_Step := ST110_Feeder_e.START;
            //STEP / END / LEERFAHREN restart
        ELSIF (enIN_State < StateAUTO) AND (enIN_State >= enState.StateSTEP) AND xIN_RestartCYCL AND NOT fifo.IsFull()
            THEN
            iOUT_Step := ST110_Feeder_e.START;
            //STEP / END / LEERFAHREN fertig
        ELSIF (enIN_State = StateREADY) THEN
            iOUT_Step := ST110_Feeder_e.READY;
        END_IF;
    END_IF;

(************ ERROR *************)
ST110_Feeder_e.ERROR: (* ERROR *) ;

END_CASE;

END_FUNCTION_BLOCK

// ---- POUs/20_AUTO/ST110/POU_ALARM_110.TcPOU
PROGRAM POU_ALARM_110
VAR_INPUT
    xIN_QUIT      : BOOL; // Alarm quittieren
    iIN_ArraySize : INT;
    pstrIN_ALARM  : POINTER TO structAlarm;       // Array Alarmstruktur
    refPOU        : REFERENCE TO FB_AUT_ABSTRACT; // the POU to test
END_VAR
VAR_OUTPUT
    xOUT_AL_ST : BOOL; // Alarm Station aktiv
END_VAR
VAR
    //Alarmbaustein
    _FB_ALARM_ST : FB_ALARM;
    //Local
    iIndex : INT; // Index For Schleife	
END_VAR
VAR CONSTANT
    sDefString : STRING := 'Error ST110,'; // Station #
END_VAR

(********************** INITIALISIERE VARIABLEN ****************************)
FOR iIndex := 0 TO iIN_ArraySize - 1 DO
    pstrIN_ALARM[iIndex].xAlarmIN   := FALSE;
    pstrIN_ALARM[iIndex].xAlarmOFF  := FALSE;
    pstrIN_ALARM[iIndex].xAlarmSAVE := TRUE;
    pstrIN_ALARM[iIndex].xAlarmQUIT := xIN_QUIT;
    pstrIN_ALARM[iIndex].tAlarmVERZ := T#100MS;
    pstrIN_ALARM[iIndex].sAlarmText := '';
    pstrIN_ALARM[iIndex].bAlarmNr   := 0;
END_FOR

(********************** ALARME ****************************)
pstrIN_ALARM[0].xAlarmIN   := (refPOU.bOUT_ErrorNum = ST110_Alarm_e.Axis_110_01Y_error);
pstrIN_ALARM[0].sAlarmText := CONCAT(sDefString, ' Axis 01Y in error');
pstrIN_ALARM[0].bAlarmNr   := 0;

pstrIN_ALARM[1].xAlarmIN   := (refPOU.bOUT_ErrorNum = ST110_Alarm_e.Axis_110_02Z_error);
pstrIN_ALARM[1].sAlarmText := CONCAT(sDefString, ' Axis 02Z (left) in error');
pstrIN_ALARM[1].bAlarmNr   := 0;

pstrIN_ALARM[2].xAlarmIN   := (refPOU.bOUT_ErrorNum = ST110_Alarm_e.Axis_110_03Z_error);
pstrIN_ALARM[2].sAlarmText := CONCAT(sDefString, ' Axis 03Z (right) in error');
pstrIN_ALARM[2].bAlarmNr   := 0;

pstrIN_ALARM[3].xAlarmIN   := (refPOU.bOUT_ErrorNum = ST110_Alarm_e.Axis_110_04Z_error);
pstrIN_ALARM[3].sAlarmText := CONCAT(sDefString, ' Axis 04Z in error');
pstrIN_ALARM[3].bAlarmNr   := 0;

pstrIN_ALARM[4].xAlarmIN   := (refPOU.bOUT_ErrorNum = ST110_Alarm_e.Cylinder_vacuum_griper_left);
pstrIN_ALARM[4].sAlarmText := CONCAT(sDefString, ' Cylinder .05 vacuum gripper right');
pstrIN_ALARM[4].bAlarmNr   := 0;

pstrIN_ALARM[5].xAlarmIN   := (refPOU.bOUT_ErrorNum = ST110_Alarm_e.Cylinder_vacuum_griper_right);
pstrIN_ALARM[5].sAlarmText := CONCAT(sDefString, ' Cylinder .06 vacuum gripper left');
pstrIN_ALARM[5].bAlarmNr   := 0;

pstrIN_ALARM[6].xAlarmIN   := (refPOU.bOUT_ErrorNum = ST110_Alarm_e.Axis_110_10W_error);
pstrIN_ALARM[6].sAlarmText := CONCAT(sDefString, ' Axis 10W in error');
pstrIN_ALARM[6].bAlarmNr   := 0;

pstrIN_ALARM[7].xAlarmIN   := (refPOU.bOUT_ErrorNum = ST110_Alarm_e.Feeder_error);
pstrIN_ALARM[7].sAlarmText := CONCAT(sDefString, ' One part of the feeder is in error');
pstrIN_ALARM[7].bAlarmNr   := 0;

pstrIN_ALARM[8].xAlarmIN   := (refPOU.bOUT_ErrorNum = ST110_Alarm_e.Piece_in_unused_griper);
pstrIN_ALARM[8].sAlarmText := CONCAT(sDefString, ' One part is handled by a unused griper');
pstrIN_ALARM[8].bAlarmNr   := 0;

pstrIN_ALARM[9].xAlarmIN   := (refPOU.bOUT_ErrorNum = ST110_Alarm_e.Piece_missing_left_griper);
pstrIN_ALARM[9].sAlarmText := CONCAT(sDefString, ' A piece is missing in the left griper');
pstrIN_ALARM[9].bAlarmNr   := 0;

pstrIN_ALARM[10].xAlarmIN   := (refPOU.bOUT_ErrorNum = ST110_Alarm_e.Piece_missing_right_griper);
pstrIN_ALARM[10].sAlarmText := CONCAT(sDefString, ' A piece is missing in the right griper');
pstrIN_ALARM[10].bAlarmNr   := 0;

pstrIN_ALARM[11].xAlarmIN   := (refPOU.bOUT_ErrorNum = ST110_Alarm_e.Feeder_empty);
pstrIN_ALARM[11].sAlarmText := CONCAT(sDefString, ' The feeder is empty');
pstrIN_ALARM[11].bAlarmNr   := 0;

pstrIN_ALARM[12].xAlarmIN   := (refPOU.bOUT_ErrorNum = ST110_Alarm_e.Reach_end_pos_without_needed_torque);
pstrIN_ALARM[12].sAlarmText := CONCAT(sDefString, ' Verticals have reached the end position without measuring the necessary torque');
pstrIN_ALARM[12].bAlarmNr   := 0;

(********************** ALARM FB ****************************)
_FB_ALARM_ST(pstrIN_Alarm  := pstrIN_ALARM,
             iIN_ArraySize := ST110_Alarm_e._max);

(********************** ALARM FB ****************************)
xOUT_AL_ST := FALSE;

FOR iIndex := 0 TO iIN_ArraySize - 1 DO
    IF pstrIN_ALARM[iIndex].xAlarmOUT THEN
        xOUT_AL_ST := TRUE;
    END_IF
END_FOR

END_PROGRAM

// ---- POUs/20_AUTO/ST115/FB_AUT_115.TcPOU
FUNCTION_BLOCK FB_AUT_115 EXTENDS FB_AUT_ABSTRACT
(****************************************************************************)
(*	POU_AUT_zxx			Bausteinaufrufe Station	zxx							*)
(*	Status				ungetestet											*)
(*  Version:			1.0													*)
(*	Beschrieb:																*)
(*																			*)
(*	Abläufe:			FB_ABLzxxA		Hauptablauf							*)
(*																			*)
(*																			*)
(* 	25.09.2019/Dj															*)
(****************************************************************************)
(*	dd.mm.yyyy   KZ    x.y			Beschrieb								*)
(****************************************************************************)
VAR_INPUT
    (* spezifische Eingänge *)

END_VAR
VAR_OUTPUT
    (* spezifische Ausgänge *)

END_VAR
VAR
    (* Bausteine *)
    fb_Pnp    : FB_ABL_115_Pnp;
    fb_Feeder : FB_ABL_115_Feeder;

    fb_stat_pnp    : FB_AUT_Statistics;
    fb_stat_Feeder : FB_AUT_Statistics;
END_VAR

VAR CONSTANT
    ROT_TABLE_FREE_MAX_Y : REAL := 200.0; // If Y and Z axis is more than this value, the feeder cannot move
    ROT_TABLE_FREE_MAX_Z : REAL := 200.0; // If Z and Y axis is more than this value, the feeder cannot move
END_VAR

(*******************************************************************)
(* Timer *)
(*******************************************************************)

(*******************************************************************)
(* Flanken / Merker *)
(*******************************************************************)
//MANU CYCLE
IF (enIN_State = StateMANU) AND xIN_ManuCycle THEN
    xManuCycle := TRUE;
END_IF;

IF (enIN_State <> StateMANU) OR xOUT_Done THEN
    xManuCycle := FALSE;
END_IF

//NEXT STEP
xNextStep := (enIN_State > StateSTEP) OR
             ((enIN_State = StateSTEP) AND xIN_Step) OR
             ((enIN_State = StateMANU) AND xManuCycle);

//RESET
xReset := (enIN_State < StateREADY) AND (enIN_State <> StateINIT) AND NOT xManuCycle;

(*******************************************************************)
(* Bausteinaufrufe Abläufe *)
(*******************************************************************)

xRelease := MAIN.MoverMan.IsProcessUsed(THIS^);

fb_Pnp(xIN_Reset          := xReset,
       xIN_Init           := xIN_Init,
       xIN_Quit           := xIN_Quit,
       xIN_Start          := enIN_State >= enState.StateLEER AND xRelease,
       xIN_Sperre         := NOT xIN_On,
       xIN_NextStep       := xNextStep,
       xIN_AlarmAktiv     := xIN_AlarmAktiv,
       xIN_DryCycle       := xIN_DryCycle,
       xIN_RestartCYCL    := enIN_State >= enState.StateLEER,
       enIN_State         := enIN_State,
       tIN_Timeout        := tIN_Timeout,
       pxFG_Freigabe      := ADR(xRelease),
       Mover              := THIS^.Mover,
       xIN_PceReadyToPick := fb_Feeder.xOUT_Done);

fb_Feeder(xIN_Reset       := xReset,
          xIN_Init        := xIN_Init,
          xIN_Quit        := xIN_Quit,
          xIN_Start       := enIN_State >= enState.StateLEER AND xRelease,
          xIN_Sperre      := NOT xIN_On,
          xIN_NextStep    := xNextStep,
          xIN_AlarmAktiv  := xIN_AlarmAktiv,
          xIN_DryCycle    := xIN_DryCycle,
          xIN_RestartCYCL := enIN_State >= enState.StateLEER,
          enIN_State      := enIN_State,
          tIN_Timeout     := tIN_Timeout,
          pxFG_Freigabe   := ADR(xRelease),
          // special
          xIN_PickPiece            := fb_Pnp.xOUT_PickPiece,
          xIN_RotTableBlockedByPnp := (ST115_Axis.axis115_01Y.rActPos > ROT_TABLE_FREE_MAX_Y) AND
                                      (ST115_Axis.axis115_02Z.rActPos > ROT_TABLE_FREE_MAX_Z));

fb_stat_pnp(xIN_Enable  := enState.StateAUTO = enIN_State,
            xIN_Waiting := fb_Pnp.xOUT_Wait,
            xIN_Running := (fb_Pnp.iOUT_Step >= ST115_Pnp_e.START) AND
                           (fb_Pnp.iOUT_Step <= ST115_Pnp_e.DONE),
            // Since we use a mover system, a cycle is done when we are waiting on a mover
            xIN_Done := fb_Pnp.iOUT_Step = ST115_Pnp_e.waitOnMover);

fb_stat_Feeder(xIN_Enable  := enState.StateAUTO = enIN_State,
               xIN_Waiting := fb_feeder.xOUT_Wait,
               xIN_Running := (fb_feeder.iOUT_Step >= ST115_Feeder_e.START) AND
                              (fb_feeder.iOUT_Step <= ST115_Feeder_e.DONE),
               xIN_Done := fb_feeder.iOUT_Step = ST115_Feeder_e.DONE);

(*******************************************************************)
(* Mover reset flags *)
(*******************************************************************)

(*******************************************************************)
(* OUTPUT *)
(*******************************************************************)
xOUT_InitDone := fb_Pnp.xOUT_InitDone AND fb_Feeder.xOUT_InitDone;
xOUT_Ready    := fb_Pnp.xOUT_Ready AND fb_Feeder.xOUT_Ready;
xOUT_Done     := fb_Pnp.xOUT_Done AND fb_Feeder.xOUT_Done;
xOUT_ErrFlag  := fb_Pnp.xOUT_ErrFlag OR fb_Feeder.xOUT_ErrFlag;
xOUT_Wait     := fb_Pnp.xOUT_Wait OR fb_Feeder.xOUT_Wait;
xOUT_AlarmST  := xOUT_ErrFlag;

(*******************************************************************)
(* Bausteinaufruf Error Station *)
(*******************************************************************)
// POU_ERR_VORLAGE(xIN_QUIT:=xIN_Quit , pstrArIN_ALARM:=ADR(HMI.strArALARM[1]));

(* % of completion of the process *)
PROPERTY iCompletionPC : INT
GET
iCompletionPC := THIS^.fb_Pnp.iOUT_ProcessCompletion;
END_GET
END_PROPERTY

PROPERTY ProcessExecution : ProcessExecution_e
GET
ProcessExecution := THIS^._ProcessExecution;
END_GET
SET
THIS^._ProcessExecution := ProcessExecution;
END_SET
END_PROPERTY

PROPERTY xBusy : BOOL
GET
xBusy := THIS^.fb_Pnp.xOUT_Busy;
END_GET
SET
END_SET
END_PROPERTY

PROPERTY xDone : BOOL
GET
xDone := THIS^.fb_Pnp.xOUT_Ready OR THIS^.fb_Pnp.xOUT_Done;
END_GET
END_PROPERTY

PROPERTY xMoverPathFree : BOOL
GET
xMoverPathFree := THIS^.fb_Pnp.xOUT_MoverFree OR THIS^.fb_Pnp.xOUT_Ready OR THIS^.fb_Pnp.xOUT_Done;
END_GET
END_PROPERTY

PROPERTY xMoverShouldLeave : BOOL
GET
xMoverShouldLeave := THIS^.fb_Pnp.iOUT_Step = ST115_Pnp_e.SYNC_MOVER_LEAVE;
END_GET
END_PROPERTY

END_FUNCTION_BLOCK

// ---- POUs/20_AUTO/ST115/FB_ABL_115_Pnp.TcPOU
FUNCTION_BLOCK FB_ABL_115_Pnp
(****************************************************************************************)
(*	TITEL				laden kristall- Modul	    										*)
(*	Status				ungetestet                         								*)
(*	Beschrieb:			Ablaufbeschreibung												*)
(*																						*)
(*	Steps:	self-explained using enum													*)
(***********************************Revisionen*******************************************)
(*	see github blames																	*)
(****************************************************************************************)

VAR_INPUT
    xIN_Reset       : BOOL;          // Schrittkette zurücksetzen 
    xIN_Init        : BOOL;          // Initialisieren
    xIN_Quit        : BOOL;          // Fehler quittieren 
    xIN_Start       : BOOL;          // Startbefehl
    xIN_Sperre      : BOOL;          // FB Sperren 
    xIN_NextStep    : BOOL;          // Nächsten Schritt ausführen 
    xIN_AlarmAktiv  : BOOL;          // Anlage hat Alarm
    xIN_DryCycle    : BOOL;          // Fahren ohne Teile
    xIN_RestartCYCL : BOOL;          // Zyklus erneut starten im STEP, END, LEERFAHREN
    enIN_State      : enState;       // Status Anlage
    tIN_Timeout     : TIME := T#10s; // Timout

    pxFG_Freigabe : POINTER TO BOOL; //Freigabe von Station

    // Application specific
    Mover              : REFERENCE TO FB_Mover;
    xIN_PceReadyToPick : BOOL; // the piece(s) is/are ready to picked
END_VAR
VAR_OUTPUT
    (* standart Ausgänge *)
    xOUT_ErrFlag  : BOOL;        // Error Flag 
    xOUT_Busy     : BOOL;        // Baustein befindet sich im Ablauf 
    xOUT_Done     : BOOL;        // Baustein hat den Ablauf beendet 		
    xOUT_Ready    : BOOL;        // Ready to begin, should be the same state as done	
    xOUT_Timeout  : BOOL;        // Timeout FB 
    xOUT_InitDone : BOOL;        // initialisierung fertig
    xOUT_Wait     : BOOL;        // Wartet auf Bedingung
    iOUT_Step     : ST115_Pnp_e; // Aktueller Schritt 
    sOUT_Step     : STRING;      // Aktueller Schritt but in string format
    bOUT_Error    : BYTE;        // Fehlernummer

    iOUT_ProcessCompletion : INT;  //process completion, express in % (0-100)
    xOUT_MoverFree         : BOOL; // The mover is free to move
    xOUT_PickPiece         : BOOL; // Set to true when a piece is picked

END_VAR
VAR
    (* Standard *)
    (* Schritt *)
    iLastStep : ST115_Pnp_e; // Merker letzter Schritt 
    iPreStep  : ST115_Pnp_e; // Schritt zurück nach Alarm 
    iAktStep  : ST115_Pnp_e; // aktueller Schritt

    // Trigger Starten 
    rtSTART : R_TRIG;
    // Timer TimeOut 
    TON_Timeout : TON;

    (* Bausteine *)

    (* Spezial *)
    fb_axis115_01Y : FB_AxisLM_V1_1;
    fb_axis115_02Z : FB_AxisLIN_V1_1;
    fb_axis115_03Z : FB_AxisLIN_V1_1;
    fb_axis115_04Z : FB_AxisLIN_V1_1;

    fb_PnpHorAxis  : FB_LinearMotionMan;
    fb_PnpVerAxisL : FB_LinearMotionMan;
    fb_PnpVerAxisR : FB_LinearMotionMan;
    fb_PnpVerAxisU : FB_LinearMotionMan;

    fb_simu_axis115_01Y : FB_Simu_AxisLM_V1_1;
    fb_simu_axis115_02Z : FB_Simu_AxisLIN_V1_1;
    fb_simu_axis115_03Z : FB_Simu_AxisLIN_V1_1;
    fb_simu_axis115_04Z : FB_Simu_AxisLIN_V1_1;
	
    fb_gripperLeft    : FB_ZylMo2El_V2_1;
    simu_gripperLeft  : FB_Simu_Zyl2Pos;
    fb_gripperRight   : FB_ZylMo2El_V2_1;
    simu_gripperRight : FB_Simu_Zyl2Pos;

END_VAR
VAR CONSTANT
    PNP_SIMULATION : BOOL := TRUE; // Set to TRUE to simulate this part of the program
END_VAR

(*******************************************************************)
(* Trigger  *)
(*******************************************************************)
(* Zurücksetzen *)
IF xIN_RESET THEN
    iPreStep  := ST115_Pnp_e.RESET;
    iOUT_Step := ST115_Pnp_e.RESET;
END_IF;

(* Error Quittieren *)
IF (bOUT_Error <> 0) AND xIN_Quit THEN
    xOUT_ErrFlag := FALSE;
    bOUT_Error   := 0;
    iOUT_Step    := iPreStep;
END_IF;

(*******************************************************************)
(* Timer *)
(*******************************************************************)
TON_Timeout(IN := xIN_NextStep AND (iLastStep = iOUT_Step) (*todo FG *) ,
            PT := tIN_Timeout);

(*******************************************************************)
(* Bausteine *)
(*******************************************************************)
fb_PnpHorAxis(config          := _20_AUTO.recipe.linearAxis[LinearAxis_e.ST115_01Y],
              xIN_Init        := enIN_State = enState.StateINIT,
              xIN_Reset       := xIN_Reset,
              lrIN_CurrPos    := fb_axis115_01Y.rOUT_ActPos,
              lrIN_Delta_mm   := 0.01,
              iIN_CurrentStep := iOUT_Step,
              iIN_moveNumber  := ST115_PnpHorPos_e._max);

fb_simu_axis115_01Y(xIN_Enable          := PNP_SIMULATION AND CONST.USE_SIMULATION,
                    bIN_AxisCntr        := fb_axis115_01Y.bOUT_AxisCntr,
                    wIN_AxisState       := ST115_Axis.axis115_01Y.wState,
                    udiIN_HomingTime_ms := 2000,
                    pIN_axisSimu        := ADR(SIMU.axis_ref[Axis_e.ST115_01Y]),
                    pIN_axisHW          := ADR(ST115_Axis.axis115_01Y.axis),
                    rIN_PosActual       := fb_axis115_01Y.rOUT_ActPos,
                    rIN_PosMax          := ST115_Axis.const115_01Y.POS_MAX,
                    rIN_PosMin          := ST115_Axis.const115_01Y.POS_MIN,
                    rIN_PixMax          := 100,
                    rIN_PixMin          := 0);

fb_axis115_01Y(enIN_State       := enIN_State,
               parIN_Buttons    := ADR(AXIS.btTeachArAxis[Axis_e.ST115_01Y]),
               xIN_DisButtons   :=,
               xIN_Quit         := xIN_Quit,
               xIN_PARAMok      := TRUE, (*TODO*)
               xIN_FREE         := TRUE,
               xIN_FREE_HOME    := TRUE,
               rIN_POSMIN       := ST115_Axis.const115_01Y.POS_MIN,
               rIN_POSMAX       := ST115_Axis.const115_01Y.POS_MAX,
               rIN_VELOMAX      := ST115_Axis.const115_01Y.VELO_MAX,
               rIN_VELOMANU     := ST115_Axis.const115_01Y.VELO_MANU,
               rIN_VELOOPEN     := ST115_Axis.const115_01Y.VELO_MANU / 4,
               rIN_JogInc       := AXIS.rTeachIncAxis,
               xIN_Execute      := fb_PnpHorAxis.xOUT_Execute,
               xIN_Home         := ST115_Pnp_e.Init_HomeHorizontals = iAktStep,
               xIN_Relative     :=,
               rIN_Position     := TO_REAL(fb_PnpHorAxis.OUT_MoveProfile.lrPosition),
               rIN_Velocity     := TO_REAL(fb_PnpHorAxis.OUT_MoveProfile.lrVelocity),
               rIN_Acceleration := TO_REAL(fb_PnpHorAxis.OUT_MoveProfile.lrAccel),
               rIN_Deceleration := TO_REAL(fb_PnpHorAxis.OUT_MoveProfile.lrDecel),
               rIN_Jerk         := TO_REAL(fb_PnpHorAxis.OUT_MoveProfile.lrJerk),
               rIN_PosManu      :=
               TO_REAL(_20_AUTO.recipe
                           .linearAxis[LinearAxis_e.ST115_01Y].movesList[AXIS.bTeachPos[Axis_e.ST115_01Y]].lrPosition),
               rIN_VeloJogManu := TO_REAL(Axis.rJogVelo_pc),
               xIN_Reset       := (ST115_Pnp_e.RESET = iOUT_Step) OR xIN_Reset,
               // the simu fb gives the hardware signal when the simulation is disabled
               wAxisState    := fb_simu_axis115_01Y.wOUT_AxisState,
               bOUT_AxisCntr => ST115_Axis.axis115_01Y.bCtrlHi,
               rOUT_ActPos   => ST115_Axis.axis115_01Y.rActPos,
               axisIN_REF    := fb_simu_axis115_01Y.pOUT_axisRef^);

fb_PnpVerAxisL(config          := _20_AUTO.recipe.linearAxis[LinearAxis_e.ST115_02Z],
               xIN_Init        := enIN_State = enState.StateINIT,
               xIN_Reset       := xIN_Reset,
               lrIN_CurrPos    := fb_axis115_02Z.rOUT_ActPos,
               lrIN_Delta_mm   := 0.01,
               iIN_CurrentStep := iOUT_Step,
               iIN_moveNumber  := ST115_PnpVerPos_e._max);

fb_simu_axis115_02Z(xIN_InSimu    := PNP_SIMULATION AND CONST.USE_SIMULATION,
                    rIN_PosActual := fb_axis115_02Z.rOUT_ActPos,
                    pIN_axisSimu  := ADR(SIMU.axis_ref[Axis_e.ST115_02Z]),
                    pIN_axisHW    := ADR(ST115_Axis.axis115_02Z.axis),
                    rIN_PosMax    := ST115_Axis.const115_02Z.POS_MAX,
                    rIN_PosMin    := ST115_Axis.const115_02Z.POS_MIN,
                    rIN_PixMax    := 80,
                    rIN_PixMin    := 0);

fb_axis115_02Z(enIN_State      := enIN_State,
               parIN_Buttons   := ADR(AXIS.btTeachArAxis[Axis_e.ST115_02Z]),
               xIN_DisButtons  :=,
               xIN_Quit        := xIN_Quit,
               xIN_AX5000      := FALSE,
               xIN_ENC_ABS     := TRUE, // TODO set accordingly
               xIN_PARAMok     := TRUE,
               xIN_FREE        := TRUE,
               xIN_FREE_HOME   := TRUE,
               rIN_POSMIN      := ST115_Axis.const115_02Z.POS_MIN,
               rIN_POSMAX      := ST115_Axis.const115_02Z.POS_MAX,
               rIN_VELOMAX     := ST115_Axis.const115_02Z.VELO_MAX,
               rIN_VELOMANU    := ST115_Axis.const115_02Z.VELO_MANU,
               rIN_VELOOPEN    := ST115_Axis.const115_02Z.POS_MAX / 4,
               rIN_JogInc      := AXIS.rTeachIncAxis,
               rIN_VeloJogManu := TO_REAL(AXIS.rJogVelo_pc),
               xIN_HomeExe     :=,
               xIN_HomeCalib   :=,
               xIN_Execute     := (_20_AUTO.recipe.st115.xUseVerLeft OR (iOUT_Step < ST115_Pnp_e.READY)) AND
                                  (fb_PnpVerAxisL.xOUT_Execute),
               xIN_HomeExe      := NOT CONST.USE_SIMULATION AND (ST115_Pnp_e.Init_HomeVerticals = iAktStep),
               xIN_Relative     :=,
               rIN_Position     := TO_REAL(fb_PnpVerAxisL.OUT_MoveProfile.lrPosition),
               rIN_Velocity     := TO_REAL(fb_PnpVerAxisL.OUT_MoveProfile.lrVelocity),
               rIN_Acceleration := TO_REAL(fb_PnpVerAxisL.OUT_MoveProfile.lrAccel),
               rIN_Deceleration := TO_REAL(fb_PnpVerAxisL.OUT_MoveProfile.lrDecel),
               rIN_Jerk         := TO_REAL(fb_PnpVerAxisL.OUT_MoveProfile.lrJerk),
               rIN_PosManu      :=
               TO_REAL(_20_AUTO.recipe
                           .linearAxis[LinearAxis_e.ST115_02Z].movesList[AXIS.bTeachPos[Axis_e.ST115_02Z]].lrPosition),
               xIN_Reset := (ST115_Pnp_e.RESET = iAktStep) OR xIN_Reset,
               // output
               rOUT_ActPos => ST115_Axis.axis115_02Z.rActPos,
               axisIN_REF  := fb_simu_axis115_02Z.pOUT_axisRef^);

fb_PnpVerAxisR(config          := _20_AUTO.recipe.linearAxis[LinearAxis_e.ST115_03Z],
               xIN_Init        := enIN_State = enState.StateINIT,
               xIN_Reset       := xIN_Reset,
               lrIN_CurrPos    := fb_axis115_03Z.rOUT_ActPos,
               lrIN_Delta_mm   := 0.01,
               iIN_CurrentStep := iOUT_Step,
               iIN_moveNumber  := ST115_PnpVerPos_e._max);

fb_simu_axis115_03Z(xIN_InSimu    := PNP_SIMULATION AND CONST.USE_SIMULATION,
                    rIN_PosActual := fb_axis115_03Z.rOUT_ActPos,
                    rIN_PosMax    := ST115_Axis.const115_03Z.POS_MAX,
                    rIN_PosMin    := ST115_Axis.const115_03Z.POS_MIN,
                    pIN_axisSimu  := ADR(SIMU.axis_ref[Axis_e.ST115_03Z]),
                    pIN_axisHW    := ADR(ST115_Axis.axis115_03Z.axis),
                    rIN_PixMax    := 80,
                    rIN_PixMin    := 0);

fb_axis115_03Z(enIN_State     := enIN_State,
               parIN_Buttons  := ADR(AXIS.btTeachArAxis[Axis_e.ST115_03Z]),
               xIN_DisButtons :=,
               xIN_Quit       := xIN_Quit,
               xIN_PARAMok    := TRUE, (*TODO*)
               xIN_FREE       := TRUE,
               xIN_FREE_HOME  := TRUE,
               rIN_POSMIN     := ST115_Axis.const115_03Z.POS_MIN,
               rIN_POSMAX     := ST115_Axis.const115_03Z.POS_MAX,
               rIN_VELOMAX    := ST115_Axis.const115_03Z.VELO_MAX,
               rIN_VELOMANU   := ST115_Axis.const115_03Z.VELO_MANU,
               rIN_VELOOPEN   := ST115_Axis.const115_03Z.VELO_MANU / 4,
               rIN_JogInc     := AXIS.rTeachIncAxis,
               xIN_Execute    := (_20_AUTO.recipe.st115.xUseVerRight OR (iOUT_Step < ST115_Pnp_e.READY)) AND
                                 (fb_PnpVerAxisR.xOUT_Execute),
               xIN_HomeExe      := NOT CONST.USE_SIMULATION AND (ST115_Pnp_e.Init_HomeVerticals = iAktStep),
               xIN_Relative     :=,
               rIN_Position     := TO_REAL(fb_PnpVerAxisR.OUT_MoveProfile.lrPosition),
               rIN_Velocity     := TO_REAL(fb_PnpVerAxisR.OUT_MoveProfile.lrVelocity),
               rIN_Acceleration := TO_REAL(fb_PnpVerAxisR.OUT_MoveProfile.lrAccel),
               rIN_Deceleration := TO_REAL(fb_PnpVerAxisR.OUT_MoveProfile.lrDecel),
               rIN_Jerk         := TO_REAL(fb_PnpVerAxisR.OUT_MoveProfile.lrJerk),
               rIN_PosManu      :=
               TO_REAL(_20_AUTO.recipe
                           .linearAxis[LinearAxis_e.ST115_03Z].movesList[AXIS.bTeachPos[Axis_e.ST115_03Z]].lrPosition),
               xIN_Reset   := (ST115_Pnp_e.RESET = iAktStep) OR xIN_Reset,
               xIN_AX5000  := FALSE,
               xIN_ENC_ABS := TRUE,
               rOUT_ActPos => ST115_Axis.axis115_03Z.rActPos, // TODO set accordingl
               axisIN_REF  := fb_simu_axis115_03Z.pOUT_axisRef^);
			   
fb_PnpVerAxisU(config          := _20_AUTO.recipe.linearAxis[LinearAxis_e.ST115_04Z],
               xIN_Init        := enState.StateINIT = enIN_State,
               xIN_Reset       := xIN_Reset,
               lrIN_CurrPos    := ST115_Axis.axis115_04Z.rActPos,
               lrIN_Delta_mm   := 0.5,
               iIN_CurrentStep := iOUT_Step,
               iIN_moveNumber  := ST115_PnpVerPushPos_e._max);

fb_simu_axis115_04Z(xIN_InSimu    := PNP_SIMULATION AND CONST.USE_SIMULATION,
                    rIN_PosActual := ST115_Axis.axis115_04Z.rActPos,
                    pIN_axisSimu  := ADR(SIMU.axis_ref[Axis_e.ST115_04Z]),
                    pIN_axisHW    := ADR(ST115_Axis.axis115_04Z.axis),
                    rIN_PosMax    := ST115_Axis.const115_04Z.POS_MAX,
                    rIN_PosMin    := ST115_Axis.const115_04Z.POS_MIN,
                    rIN_PixMax    := 80,
                    rIN_PixMin    := 0);

fb_axis115_04Z(enIN_State       := enIN_State,
               parIN_Buttons    := ADR(AXIS.btTeachArAxis[Axis_e.ST115_04Z]),
               xIN_DisButtons   :=,
               xIN_Quit         := xIN_Quit,
               xIN_AX5000       := TRUE,
               xIN_ENC_ABS      := TRUE,
               xIN_PARAMok      := TRUE,
               xIN_FREE         := TRUE,
               xIN_FREE_HOME    := TRUE,
               rIN_POSMIN       := ST115_Axis.const115_04Z.POS_MIN,
               rIN_POSMAX       := ST115_Axis.const115_04Z.POS_MAX,
               rIN_VELOMAX      := ST115_Axis.const115_04Z.VELO_MAX,
               rIN_VELOMANU     := ST115_Axis.const115_04Z.VELO_MANU,
               rIN_VELOOPEN     := ST115_Axis.const115_04Z.VELO_MANU / 4,
               rIN_JogInc       := AXIS.rTeachIncAxis,
               rIN_VeloJogManu  := TO_REAL(AXIS.rJogVelo_pc),
               xIN_HomeExe      :=,
               xIN_HomeCalib    := FALSE,
               xIN_Execute      := fb_PnpVerAxisU.xOUT_Execute,
               xIN_Relative     := FALSE,
               rIN_Position     := LREAL_TO_REAL(fb_PnpVerAxisU.OUT_MoveProfile.lrPosition),
               rIN_Velocity     := LREAL_TO_REAL(fb_PnpVerAxisU.OUT_MoveProfile.lrVelocity),
               rIN_Acceleration := LREAL_TO_REAL(fb_PnpVerAxisU.OUT_MoveProfile.lrAccel),
               rIN_Deceleration := LREAL_TO_REAL(fb_PnpVerAxisU.OUT_MoveProfile.lrDecel),
               rIN_Jerk         := LREAL_TO_REAL(fb_PnpVerAxisU.OUT_MoveProfile.lrJerk),
               rIN_PosManu      :=
               TO_REAL(_20_AUTO.recipe
                           .linearAxis[LinearAxis_e.ST115_04Z].movesList[AXIS.bTeachPos[Axis_e.ST115_04Z]].lrPosition),
               xIN_Reset   := xIN_Reset,
               rOUT_ActPos => ST115_Axis.axis115_04Z.rActPos,
               axisIN_REF  := fb_simu_axis115_04Z.pOUT_axisRef^);

// pneumatics
fb_gripperLeft(xIN_Reset    := xIN_Reset OR (ST115_Pnp_e.RESET = iOUT_Step),
               xIN_Quit     := xIN_Quit,
               xIN_Manu     := enState.StateMANU = enIN_State,
               pbtIN_Button := ADR(HMI.btManuCylinders[StationList_e.ST115][1]),
               xIN_GS       := simu_gripperLeft.xOUT_inGS,
               xIN_AS       := simu_gripperLeft.xOUT_inAS,
               xIN_FREE     := TRUE,
               xINtoGS      := ST115_Pnp_e.Gripper_close = iOUT_Step,
               xINtoAS      := _20_AUTO.recipe.st115.xUseVerLeft AND (ST115_Pnp_e.Gripper_open = iOUT_Step),
               tIN_ErrAS    := DINT_TO_TIME(_20_AUTO.recipe.cylinder2Pos[StationList_e.ST115]
                                                [ST115_Cylinders_e.GreiferLinks].toAS_alarm_time),
               tIN_ErrGS := DINT_TO_TIME(_20_AUTO.recipe.cylinder2Pos[StationList_e.ST115]
                                             [ST115_Cylinders_e.GreiferLinks].toGS_alarm_time),
               tIN_WaitAS := DINT_TO_TIME(_20_AUTO.recipe.cylinder2Pos[StationList_e.ST115]
                                              [ST115_Cylinders_e.GreiferLinks].toAS_wait_time),
               tIN_WaitGS := DINT_TO_TIME(_20_AUTO.recipe.cylinder2Pos[StationList_e.ST115]
                                              [ST115_Cylinders_e.GreiferLinks].toGS_wait_time));

simu_gripperLeft(xIN_Enable := PNP_SIMULATION AND CONST.USE_SIMULATION,
                 xIN_inGS   := IO_BOX.I6100_ST115_greifer_links_offen,
                 xIN_inAS   := IO_BOX.I6101_ST115_greifer_links_geschlossen,
                 xIN_valve  := fb_gripperLeft.xOUT_VALVE,
                 tIN_GS_ms  := 200,  //ms
                 tIN_AS_ms  := 200); //ms

fb_gripperRight(xIN_Reset    := xIN_Reset OR (ST115_Pnp_e.RESET = iOUT_Step),
                xIN_Quit     := xIN_Quit,
                xIN_Manu     := enState.StateMANU = enIN_State,
                pbtIN_Button := ADR(HMI.btManuCylinders[StationList_e.ST115][2]),
                xIN_GS       := simu_gripperRight.xOUT_inGS,
                xIN_AS       := simu_gripperRight.xOUT_inAS,
                xIN_FREE     := TRUE,
                xINtoGS      := ST115_Pnp_e.Gripper_close = iOUT_Step,
                xINtoAS      := _20_AUTO.recipe.st115.xUseVerRight AND (ST115_Pnp_e.Gripper_open = iOUT_Step),
                tIN_ErrAS    := DINT_TO_TIME(_20_AUTO.recipe.cylinder2Pos[StationList_e.ST115]
                                                 [ST115_Cylinders_e.GreiferRechts].toAS_alarm_time),
                tIN_ErrGS := DINT_TO_TIME(_20_AUTO.recipe.cylinder2Pos[StationList_e.ST115]
                                              [ST115_Cylinders_e.GreiferRechts].toGS_alarm_time),
                tIN_WaitAS := DINT_TO_TIME(_20_AUTO.recipe.cylinder2Pos[StationList_e.ST115]
                                               [ST115_Cylinders_e.GreiferRechts].toAS_wait_time),
                tIN_WaitGS := DINT_TO_TIME(_20_AUTO.recipe.cylinder2Pos[StationList_e.ST115]
                                               [ST115_Cylinders_e.GreiferRechts].toGS_wait_time));

simu_gripperRight(xIN_Enable := PNP_SIMULATION AND CONST.USE_SIMULATION,
                  xIN_inGS   := IO_BOX.I6200_ST115_greifer_rechts_offen,
                  xIN_inAS   := IO_BOX.I6201_ST115_greifer_rechts_geschlossen,
                  xIN_valve  := fb_gripperRight.xOUT_VALVE,
                  tIN_GS_ms  := 200,  //ms
                  tIN_AS_ms  := 200); //ms

(*******************************************************************)
(* OUTPUTS *)
(*******************************************************************)
// Error Flag 
xOUT_ErrFlag := (bOUT_Error <> 0) OR (ST115_Pnp_e.ERROR = iOUT_Step);
// Baustein befindet sich im Ablauf 
xOUT_Busy := (iOUT_Step > ST115_Pnp_e.READY) AND (iOUT_Step < ST115_Pnp_e.DONE);
// Baustein hat den Ablauf beendet
xOUT_Done := (iOUT_Step = ST115_Pnp_e.DONE);
// Process ready
xOUT_Ready := (iOUT_Step = ST115_Pnp_e.READY) OR (iOUT_Step = ST115_Pnp_e.waitOnMover);
// Timeout FB 				 		
xOUT_Timeout := TON_Timeout.Q;
// Itialisierung fertig			
xOUT_InitDone := (iOUT_Step = ST115_Pnp_e.READY) OR (iOUT_Step = ST115_Pnp_e.waitOnMover);
// Aktueller Schritt			
iOUT_Step := iOUT_Step; //Im Ablauf gesetzt		
sOUT_Step := TO_STRING(iOUT_Step);
//Fehlernummer	 
bOUT_Error := bOUT_Error; //Im Ablauf/FB gesetzt	
(* Warte (alle Schritte wo auf FG oder Teile gewartet wird) *)
xOUT_Wait := (iOUT_Step = ST115_Pnp_e.DONE) OR
             (iOUT_Step = ST115_Pnp_e.READY) OR
             (iOUT_Step = ST115_Pnp_e.START) OR
             (iOUT_Step = ST115_Pnp_e.waitOnMover) OR
             (iOUT_Step = ST115_Pnp_e.SYNC_MOVER_LEAVE) OR
             (iOUT_Step = ST115_Pnp_e.PnP_WaitOnFeeder);

xOUT_MoverFree := iOUT_Step >= ST115_Pnp_e.MOVER_FREE_OP AND iOUT_Step < ST115_Pnp_e.MOVER_NEEDED_OP;

iOUT_ProcessCompletion := F_GetPercent_2(iAktStep,
                                         ST115_Pnp_e.PnP_Hor_ToRotTablePos,
                                         ST115_Pnp_e.PnP_Hor_ToTrackPos,
                                         ST115_Pnp_e.PnP_Ver_ShuttleDown,
                                         ST115_Pnp_e.PnP_Ver_ShuttleUp);

xOUT_PickPiece := iOUT_Step = ST115_Pnp_e.PnP_Hor_ToTrackPos;

(*******************************************************************)
(* Ablauf *)
(*******************************************************************)

(* Sperren *)
IF xIN_Sperre THEN
    iPreStep  := ST115_Pnp_e.RESET;
    iOUT_Step := ST115_Pnp_e.RESET;
    RETURN;
END_IF;

(* Schritt Merker *)
IF iAktStep <> iOUT_Step THEN
    iLastStep := iAktStep;
    iAktStep  := iOUT_Step;
END_IF

(* START *)
rtSTART(CLK := xIN_Start);

(*******************************************************************)
(* Schrittkette  *)
(*******************************************************************)
CASE iOUT_Step OF

(***** RESET *****)
ST115_Pnp_e.RESET: (* Schritt 0-99 *)
    //Initialisierungen
    //Start Init Ablauf
    IF xIN_Init THEN
        iOUT_Step := ST115_Pnp_e.INIT;
        //Start Manu Ablauf
    ELSIF enIN_State = StateMANU AND xIN_NextStep THEN
        iOUT_Step := ST115_Pnp_e.INIT;
    END_IF;

(***** INIT *****)
ST115_Pnp_e.INIT: (* Grundstellung ? *)
    IF CONST.USE_SIMULATION THEN
        iOUT_Step := ST115_Pnp_e.Init_VerticalsUp;
    ELSE
        iOUT_Step := ST115_Pnp_e.Init_HomeVerticals;
    END_IF;

ST115_Pnp_e.Init_HomeVerticals:
    fb_axis115_02Z.rIN_Velocity := _20_AUTO.recipe.linearAxis[LinearAxis_e.ST115_02Z].movesList[0].lrVelocity;
    fb_axis115_03Z.rIN_Velocity := _20_AUTO.recipe.linearAxis[LinearAxis_e.ST115_03Z].movesList[0].lrVelocity;

    IF fb_axis115_02Z.xOUT_DONE AND fb_axis115_03Z.xOUT_DONE THEN
        iOUT_Step := ST115_Pnp_e.Init_VerticalsUp;
    END_IF

ST115_Pnp_e.Init_VerticalsUp:
    IF fb_gripperLeft.xIN_AS OR fb_gripperRight.xIN_AS THEN
        IF fb_PnpVerAxisL.MoveTo(ST115_PnpVerPos_e.UpFull).xOUT_InPos AND
           fb_PnpVerAxisR.MoveTo(ST115_PnpVerPos_e.UpFull).xOUT_InPos THEN
            IF fb_axis115_01Y.xOUT_READY OR fb_axis115_01Y.xOUT_HOMED THEN
                iOUT_Step := ST115_Pnp_e.Init_HorizontalsToTrack;
            ELSE
                iOUT_Step := ST115_Pnp_e.Init_HomeHorizontals;
            END_IF
        END_IF
    ELSE
        IF fb_PnpVerAxisL.MoveTo(ST115_PnpVerPos_e.UpEmpty).xOUT_InPos AND
           fb_PnpVerAxisR.MoveTo(ST115_PnpVerPos_e.UpEmpty).xOUT_InPos THEN
            IF fb_axis115_01Y.xOUT_READY OR fb_axis115_01Y.xOUT_HOMED THEN
                iOUT_Step := ST115_Pnp_e.Init_HorizontalsToTrack;
            ELSE
                iOUT_Step := ST115_Pnp_e.Init_HomeHorizontals;
            END_IF
        END_IF
    END_IF

ST115_Pnp_e.Init_HomeHorizontals:
    fb_axis115_01Y.rIN_Velocity := _20_AUTO.recipe.linearAxis[LinearAxis_e.ST115_01Y].defProfile.lrVelocity;

    IF fb_axis115_01Y.xOUT_HOMED THEN
        iOUT_Step := ST115_Pnp_e.Init_HorizontalsToTrack;
    END_IF

ST115_Pnp_e.Init_HorizontalsToTrack:
    IF fb_PnpHorAxis.MoveTo(ST115_PnpHorPos_e.GS).xOUT_InPos THEN
        iOUT_Step := ST115_Pnp_e.Init_check_if_pces_handled;
    END_IF

ST115_Pnp_e.Init_check_if_pces_handled:
    IF (NOT _20_AUTO.recipe.st115.xUseVerLeft AND fb_gripperLeft.xOUT_inAS) OR
       (NOT _20_AUTO.recipe.st115.xUseVerRight AND fb_gripperRight.xOUT_inAS) THEN
        // ERROR: a piece is present in an unused gripper
        bOUT_Error := 1;
        iOUT_Step  := ST115_Pnp_e.ERROR;

    ELSIF _20_AUTO.recipe.st115.xUseVerLeft AND
          NOT fb_gripperLeft.xOUT_inAS AND
          _20_AUTO.recipe.st115.xUseVerRight AND
          fb_gripperRight.xOUT_inAS THEN
        // ERROR:  Initialisation failed. A piece is missing in the left griper.
        bOUT_Error := 2;
        iOUT_Step  := ST115_Pnp_e.ERROR;

    ELSIF _20_AUTO.recipe.st115.xUseVerLeft AND
          fb_gripperLeft.xOUT_inAS AND
          _20_AUTO.recipe.st115.xUseVerRight AND
          NOT fb_gripperRight.xOUT_inAS THEN
        // ERROR:  Initialisation failed. A piece is missing in the right griper.
        bOUT_Error := 3;
        iOUT_Step  := ST115_Pnp_e.ERROR;

    ELSIF NOT fb_gripperLeft.xOUT_inAS AND NOT fb_gripperRight.xOUT_inAS THEN
        iOUT_Step := ST115_Pnp_e.READY;

    ELSE
        iOUT_Step := ST115_Pnp_e.waitOnMover;
    END_IF

(***** READY / INIT DONE *****)
ST115_Pnp_e.READY:    (* Start AUTO,END,LEER,STEP *)
    IF xIN_Start THEN //IF rtSTART.Q THEN
        iOUT_Step := ST115_Pnp_e.START;
    END_IF

(***** START  ZYKLISCH *****)
ST115_Pnp_e.START: (*  *)
    IF xIN_NextStep AND pxFG_Freigabe^ THEN
        iOUT_Step := ST115_Pnp_e.PnP_Hor_ToRotTablePos;
    END_IF;

ST115_Pnp_e.PnP_Hor_ToRotTablePos:
    IF xIN_NextStep AND fb_PnpHorAxis.MoveTo(ST115_PnpHorPos_e.AS).xOUT_InPos THEN
        iOUT_Step := ST115_Pnp_e.PnP_WaitOnFeeder;
    END_IF

ST115_Pnp_e.PnP_WaitOnFeeder:
    IF xIN_PceReadyToPick THEN
        iOUT_Step := ST115_Pnp_e.PnP_Ver_RotTableDown;
    END_IF

ST115_Pnp_e.PnP_Ver_RotTableDown:
    IF xIN_NextStep AND
       (fb_PnpVerAxisL.MoveTo(ST115_PnpVerPos_e.DownEmpty).xOUT_InPos OR
       NOT _20_AUTO.recipe.st115.xUseVerLeft) AND
       (fb_PnpVerAxisR.MoveTo(ST115_PnpVerPos_e.DownEmpty).xOUT_InPos OR
       NOT _20_AUTO.recipe.st115.xUseVerRight) THEN
        iOUT_Step := ST115_Pnp_e.Gripper_open;
    END_IF;

ST115_Pnp_e.Gripper_open:
    IF xIN_NextStep AND
       (NOT _20_AUTO.recipe.st115.xUseVerLeft OR fb_gripperLeft.xOUT_inAS) AND
       (NOT _20_AUTO.recipe.st115.xUseVerRight OR fb_gripperRight.xOUT_inAS) THEN
        iOUT_Step := ST115_Pnp_e.PnP_Ver_RotTableUp;
    END_IF;

ST115_Pnp_e.PnP_Ver_RotTableUp:
    IF xIN_NextStep AND
       (fb_PnpVerAxisL.MoveTo(ST115_PnpVerPos_e.UpFull).xOUT_InPos OR
       NOT _20_AUTO.recipe.st115.xUseVerLeft) AND
       (
       fb_PnpVerAxisR.MoveTo(ST115_PnpVerPos_e.UpFull).xOUT_InPos OR
       NOT _20_AUTO.recipe.st115.xUseVerRight
           ) THEN
        iOUT_Step := ST115_Pnp_e.PnP_Hor_ToTrackPos;
    END_IF;

ST115_Pnp_e.PnP_Hor_ToTrackPos:
    IF xIN_NextStep AND fb_PnpHorAxis.MoveTo(ST115_PnpHorPos_e.GS).xOUT_InPos THEN
        iOUT_Step := ST115_Pnp_e.waitOnMover;
    END_IF

ST115_Pnp_e.waitOnMover: (*  *)
    IF xIN_NextStep AND __ISVALIDREF(Mover) THEN
        iOUT_Step := ST115_Pnp_e.PnP_Ver_ShuttleDown;
    END_IF;

ST115_Pnp_e.PnP_Ver_ShuttleDown:
    IF xIN_NextStep AND
       (fb_PnpVerAxisL.MoveTo(ST115_PnpVerPos_e.DownFullQuick).xOUT_InPos OR
       NOT _20_AUTO.recipe.st115.xUseVerLeft) AND
       (fb_PnpVerAxisR.MoveTo(ST115_PnpVerPos_e.DownFullQuick).xOUT_InPos OR
       NOT _20_AUTO.recipe.st115.xUseVerRight) THEN
        iOUT_Step := ST115_Pnp_e.PnP_Ver_ShuttleTorqueControl;
    END_IF;

// We need a fb that enables for us torque control. Here we just go a bit further
ST115_Pnp_e.PnP_Ver_ShuttleTorqueControl:
    IF xIN_NextStep AND
       (fb_PnpVerAxisL.MoveTo(ST115_PnpVerPos_e.DownFullTorqueControl).xOUT_InPos OR
       NOT _20_AUTO.recipe.st115.xUseVerLeft) AND
       (fb_PnpVerAxisR.MoveTo(ST115_PnpVerPos_e.DownFullTorqueControl).xOUT_InPos OR
       NOT _20_AUTO.recipe.st115.xUseVerRight) THEN
        iOUT_Step := ST115_Pnp_e.Gripper_close;
    END_IF;

ST115_Pnp_e.Gripper_close:
    IF xIN_NextStep AND fb_gripperLeft.xOUT_inGS AND fb_gripperRight.xOUT_inGS THEN
        iOUT_Step := ST115_Pnp_e.PnP_Ver_ShuttleUp;
    END_IF;

ST115_Pnp_e.PnP_Ver_ShuttleUp:
    IF xIN_NextStep AND
       (fb_PnpVerAxisL.MoveTo(ST115_PnpVerPos_e.UpEmpty).xOUT_InPos OR
       NOT _20_AUTO.recipe.st115.xUseVerLeft) AND
       (fb_PnpVerAxisR.MoveTo(ST115_PnpVerPos_e.UpEmpty).xOUT_InPos OR
       NOT _20_AUTO.recipe.st115.xUseVerRight) THEN
        iOUT_Step := ST115_Pnp_e.SYNC_MOVER_LEAVE;
    END_IF;

ST115_Pnp_e.SYNC_MOVER_LEAVE:
    // The mover needs to be taken by MoverMan
    IF NOT __ISVALIDREF(Mover) THEN
        iOUT_Step := ST115_Pnp_e.DONE;
    END_IF

(***** DONE *****)
ST115_Pnp_e.DONE: (* Letzter Schritt  *)
    IF NOT xIN_AlarmAktiv THEN
        //AUTO
        IF (enIN_State = StateAUTO) AND xIN_RestartCYCL THEN
            iOUT_Step := ST115_Pnp_e.START;
            //STEP / END / LEERFAHREN restart
        ELSIF (enIN_State < StateAUTO) AND (enIN_State >= enState.StateSTEP) AND xIN_RestartCYCL THEN
            iOUT_Step := ST115_Pnp_e.START;
            //STEP / END / LEERFAHREN fertig
        ELSIF (enIN_State = StateREADY) THEN
            iOUT_Step := ST115_Pnp_e.READY;
        END_IF;
    END_IF;

(************ ERROR *************)
ST115_Pnp_e.ERROR: (* ERROR *) ;

END_CASE;

END_FUNCTION_BLOCK

// ---- POUs/20_AUTO/ST115/FB_ABL_115_Feeder.TcPOU
FUNCTION_BLOCK FB_ABL_115_Feeder
(****************************************************************************************)
(*	TITEL				laden Kristall modul, Feeder and rotary table                   *)
(*	Status				ungetestet                         								*)
(*	Beschrieb:			Ablaufbeschreibung												*)
(*																						*)
(*	Steps:	self-explained using enum													*)
(***********************************Revisionen*******************************************)
(*	see github blames																	*)
(****************************************************************************************)

VAR_INPUT
    xIN_Reset       : BOOL;          // Schrittkette zurücksetzen 
    xIN_Init        : BOOL;          // Initialisieren
    xIN_Quit        : BOOL;          // Fehler quittieren 
    xIN_Start       : BOOL;          // Startbefehl
    xIN_Sperre      : BOOL;          // FB Sperren 
    xIN_NextStep    : BOOL;          // Nächsten Schritt ausführen 
    xIN_AlarmAktiv  : BOOL;          // Anlage hat Alarm
    xIN_DryCycle    : BOOL;          // Fahren ohne Teile
    xIN_RestartCYCL : BOOL;          // Zyklus erneut starten im STEP, END, LEERFAHREN
    enIN_State      : enState;       // Status Anlage
    tIN_Timeout     : TIME := T#10s; // Timout

    pxFG_Freigabe : POINTER TO BOOL; //Freigabe von Station

    // Application specific
    xIN_PickPiece : BOOL; (* signal from the pick and place element
                             the number of picked signal depend on the recipe *)
    xIN_RotTableBlockedByPnp : BOOL; // Is the pick and place blocking the rotary table?
END_VAR
VAR_OUTPUT
    (* standart Ausgänge *)
    xOUT_ErrFlag  : BOOL;           // Error Flag 
    xOUT_Busy     : BOOL;           // Baustein befindet sich im Ablauf 
    xOUT_Done     : BOOL;           // Baustein hat den Ablauf beendet 		
    xOUT_Ready    : BOOL;           // Ready to begin, should be the same state as done	
    xOUT_Timeout  : BOOL;           // Timeout FB 
    xOUT_InitDone : BOOL;           // initialisierung fertig
    xOUT_Wait     : BOOL;           // Wartet auf Bedingung
    iOUT_Step     : ST115_Feeder_e; // Aktueller Schritt 
    sOUT_Step     : STRING;         // Aktueller Schritt but in string format
    bOUT_Error    : BYTE;           // Fehlernummer

    // Application specific
    xOUT_PceReadyToPick : BOOL; // the piece(s) is/are ready to picked
END_VAR
VAR
    (* Standard *)
    (* Schritt *)
    iLastStep : ST115_Feeder_e; // Merker letzter Schritt 
    iPreStep  : ST115_Feeder_e; // Schritt zurück nach Alarm 
    iAktStep  : ST115_Feeder_e; // aktueller Schritt

    // Trigger Starten 
    rtSTART : R_TRIG;
    // Timer TimeOut 
    TON_Timeout : TON;

    (* Bausteine *)
	btfb_feeder					: FB_BUTTON;

    // Application specific
    fb_axis115_10W               : FB_AxisLMturn_V1_1;
    simu_axis115_10W             : FB_Simu_AxisLM_V1_1;
    fb_feeder                    : FB_Feeder2Sensors;
    fifo                         : FB_Fifo(3);
    simu_feeder                  : FB_Simu_Feeder; // simulation of a feeder
    simu_fifo_feeder_to_rotTable : FB_Fifo(20);    // fifo to hold a piece
    rtPutPiece                   : R_TRIG;         // trigger to add a piece

    rtPick : R_TRIG; // r_trig signal from the pick and place machine

    iCurrentTableIndex : INT; // current table index
    iSearchIndex       : INT; (* Initialization index TO see how many element we have AT startup
                                 or after an alarm *)

    tof_color_sensor : TOF;
    simu_blow        : BOOL; // todo remove when the hardware will be used

END_VAR
VAR CONSTANT
    MAX_SEARCH_TURN : INT := 3; // maximum search number

    FEEDER_SIMULATION : BOOL := TRUE; // Simulate this code
END_VAR

(*******************************************************************)
(* Trigger  *)
(*******************************************************************)
(* Zurücksetzen *)
IF xIN_RESET THEN
    iPreStep  := ST115_Feeder_e.RESET;
    iOUT_Step := ST115_Feeder_e.RESET;
END_IF;

(* Error Quittieren *)
IF (bOUT_Error <> 0) AND xIN_Quit THEN
    xOUT_ErrFlag := FALSE;
    bOUT_Error   := 0;
    iOUT_Step    := iPreStep;
END_IF;

iCurrentTableIndex := iCurrentTableIndex MOD 3;

(*******************************************************************)
(* Timer *)
(*******************************************************************)
TON_Timeout(IN := xIN_NextStep AND (iLastStep = iOUT_Step) (*todo FG *) ,
            PT := tIN_Timeout);

(*******************************************************************)
(* Bausteine *)
(*******************************************************************)
btfb_feeder(pbtIN := ADR(HMI.btManuCylinders[StationList_e.ST115][3]),
				xINdis:= (enIN_State<>enState.StateMANU),
				xINon:= ,
				xINerr:= fb_feeder.xOUT_Empty);

IF btfb_feeder.pbtIN^.rtrig THEN
	btfb_feeder.xINon := NOT btfb_feeder.xINon;
ELSIF (enIN_State<>enState.StateMANU) THEN
	btfb_feeder.xINon := FALSE;
END_IF;

fb_feeder(xIN_Enable                := ((enIN_State<=enState.StateAUTO) AND (enIN_State>=enState.StateSTEP)) 
										OR btfb_feeder.xINon,
          xIN_PieceInEnd            := IO_BOX.I6001_ST115_teil_in_vereinzelung,
          xIN_PieceMax              := IO_BOX.I8101_ST115_maximum,
          xIN_InSimulation          := FEEDER_SIMULATION AND CONST.USE_SIMULATION,
          refIN_SimulatedFifo       := simu_fifo_feeder_to_rotTable,
          iIN_FifoSetMaxSensorValue := 10,
          diIN_SignlFilter_ms       := _20_AUTO.recipe.st115.FeederConfig.InFilterDelay,
          diIN_StartDelay_ms        := _20_AUTO.recipe.st115.FeederConfig.StartDelay,
          diIN_StopDelay_ms         := _20_AUTO.recipe.st115.FeederConfig.StopDelay,
          diIN_EmptyDelay_ms        := _20_AUTO.recipe.st115.FeederConfig.EmptyDelay);

simu_feeder(xIN_Enable         := fb_feeder.xOUT_EnableFeeder AND FEEDER_SIMULATION AND CONST.USE_SIMULATION,
            xIN_PceSensor      := fb_feeder.xIN_PieceInEnd,
            tIN_NewPieceTime   := 500,
            iIN_WaitTimeMin_ms := 500,
            iIN_WaitTimeMax_ms := 1000);

rtPick(CLK := xIN_PickPiece);
rtPutPiece(CLK := simu_feeder.xOUT_NewPiece);

IF rtPutPiece.Q AND NOT simu_fifo_feeder_to_rotTable.IsFull() THEN
    simu_fifo_feeder_to_rotTable.Put(1);
END_IF

IF ST115_Feeder_e.Init_simu_home_table = iOUT_Step THEN
    fb_axis115_10W.rIN_Position := TO_REAL(120.0 - LMOD(ST115_Axis.axis115_10W.rActPos, 120.0));

ELSIF ST115_Feeder_e.Init_home_table = iOUT_Step THEN
    fb_axis115_10W.rIN_Position := TO_REAL(120.0 - LMOD(ST115_Axis.axis115_10W.rActPos, 120.0));

ELSIF ST115_Feeder_e.Init_table_go_to_zero = iOUT_Step THEN
    fb_axis115_10W.rIN_Position := 360 - ST115_Axis.axis115_10W.rActPos;

ELSE
    fb_axis115_10W.rIN_Position := 120.0;

END_IF

simu_axis115_10W(xIN_Enable          := FEEDER_SIMULATION AND CONST.USE_SIMULATION,
                 wIN_AxisState       := ST115_Axis.axis115_10W.wState,
                 bIN_AxisCntr        := fb_axis115_10W.bOUT_AxisCntr,
                 udiIN_HomingTime_ms := 1000,
                 pIN_axisSimu        := ADR(SIMU.axis_ref[Axis_e.ST115_10W]),
                 pIN_axisHW          := ADR(ST115_Axis.axis115_10W.axis),
                 rIN_PosActual       := fb_axis115_10W.rOUT_ActPos,
                 rIN_PosMax          := ST115_Axis.const115_10W.POS_MAX,
                 rIN_PosMin          := ST115_Axis.const115_10W.POS_MIN,
                 rIN_PixMax          := 0,
                 rIN_PixMin          := 0);

fb_axis115_10W(enIN_State     := enIN_State,
               parIN_Buttons  := ADR(AXIS.btTeachArAxis[Axis_e.ST115_10W]),
               xIN_DisButtons := ,
               xIN_Quit       := xIN_Quit,
               xIN_PARAMok    := TRUE,
               xIN_FREE       := NOT xIN_RotTableBlockedByPnp,
               xIN_FREE_HOME  := TRUE,
               rIN_POSMIN     := ST115_Axis.const115_10W.POS_MIN,
               rIN_POSMAX     := ST115_Axis.const115_10W.POS_MAX,
               rIN_VELOMAX    := ST115_Axis.const115_10W.VELO_MAX,
               rIN_VELOMANU   := ST115_Axis.const115_10W.VELO_MANU,
               rIN_VELOOPEN   := ST115_Axis.const115_10W.VELO_MANU / 4,
               rIN_JogInc     := AXIS.rTeachIncAxis,
               xIN_Execute    := ST115_Feeder_e.Init_set_table_pos = iOUT_Step OR
                                 ST115_Feeder_e.Init_table_go_to_zero = iOUT_Step OR
                                 ST115_Feeder_e.Init_simu_home_table = iOUT_Step OR
                                 ST115_Feeder_e.load_piece = iOUT_Step OR
                                 ST115_Feeder_e.wait_rotary_table_done = iOUT_Step,
               xIN_Relative     := fb_axis115_10W.xIN_Execute,
               xIN_STOP         := FALSE,
               xIN_OFF          := FALSE,
               rIN_Position     :=, // Is set above
               rIN_Velocity     := TO_REAL(720.0),
               rIN_Acceleration := TO_REAL(1440.0),
               rIN_Deceleration := TO_REAL(7200.0),
               rIN_Jerk         := TO_REAL(720000.0),
               xIN_Home         := ST115_feeder_e.Init_home_table = iOUT_Step,
               xIN_Reset        := xIN_Reset OR ST115_feeder_e.RESET = iOUT_Step,
               // The simu fb gives us the hardware signal when we are not in simulation
               wAxisState    := simu_axis115_10W.wOUT_AxisState,
               bOUT_AxisCntr => ST115_Axis.axis115_10W.bCtrlHi,
               rOUT_ActPos   =>, // leave empty, rActPos must be set using the modulo
               axisIN_REF    := simu_axis115_10W.pOUT_axisRef^);

ST115_Axis.axis115_10W.rActPos := LREAL_TO_REAL(simu_axis115_10W.pOUT_axisRef^.NcToPlc.ModuloActPos);

(*******************************************************************)
(* OUTPUTS *)
(*******************************************************************)
// Error Flag 
xOUT_ErrFlag := (bOUT_Error <> 0) OR (ST115_Feeder_e.ERROR = iOUT_Step);
// Baustein befindet sich im Ablauf 
xOUT_Busy := (iOUT_Step > ST115_Feeder_e.READY) AND (iOUT_Step < ST115_Feeder_e.DONE);
// Baustein hat den Ablauf beendet
xOUT_Done := (iOUT_Step = ST115_Feeder_e.DONE);
// Process ready
xOUT_Ready := (iOUT_Step = ST115_Feeder_e.READY);
// Timeout FB 				 		
xOUT_Timeout := TON_Timeout.Q;
// Itialisierung fertig			
xOUT_InitDone := (iOUT_Step = ST115_Feeder_e.READY);
// Aktueller Schritt			
iOUT_Step := iOUT_Step; //Im Ablauf gesetzt		
sOUT_Step := TO_STRING(iOUT_Step);
//Fehlernummer	 
bOUT_Error := bOUT_Error; //Im Ablauf/FB gesetzt	
(* Warte (alle Schritte wo auf FG oder Teile gewartet wird) *)
xOUT_Wait := (iOUT_Step = ST115_Feeder_e.DONE) OR
             (iOUT_Step = ST115_Feeder_e.READY);

// // TODO add simulation constant to prevent the output to be set
// IO_BOX.Q8000_ST115_freigabe_wf    := fb_feeder.xOUT_EnableFeeder; // AND SIMULATION CONSTANT
// IO_BOX.Q8003_ST115_forderband_ein :=
//     (iOUT_Step <> ST115_Feeder_e.DONE) AND NOT fb_feeder.xIN_PieceInEnd; // AND SIMULATION CONSTANT
// 
// // blow out
// tof_color_sensor(IN := IO_BOX.I8004_ST115_farbsensor_lagekontrolle,
//                  PT := DINT_TO_TIME(_20_AUTO.recipe.st115.blowPieceTof_ms));
// 
// simu_blow := tof_color_sensor.Q;

(*******************************************************************)
(* Ablauf *)
(*******************************************************************)

(* Sperren *)
IF xIN_Sperre THEN
    iPreStep  := ST115_Feeder_e.RESET;
    iOUT_Step := ST115_Feeder_e.RESET;
    RETURN;
END_IF;

(* Schritt Merker *)
IF iAktStep <> iOUT_Step THEN
    iLastStep := iAktStep;
    iAktStep  := iOUT_Step;
END_IF

(* START *)
rtSTART(CLK := xIN_Start);

(*******************************************************************)
(* Schrittkette  *)
(*******************************************************************)
CASE iOUT_Step OF

(***** RESET *****)
ST115_Feeder_e.RESET: (* Schritt 0-99 *)
    //Initialisierungen
    //Start Init Ablauf
    IF xIN_Init THEN
        iOUT_Step := ST115_Feeder_e.INIT;
        //Start Manu Ablauf
    ELSIF enIN_State = StateMANU AND xIN_NextStep THEN
        iOUT_Step := ST115_Feeder_e.INIT;
    END_IF;

(***** INIT *****)
ST115_Feeder_e.INIT: (* Grundstellung ? *)
    IF NOT xIN_RotTableBlockedByPnp THEN
        iOUT_Step := ST115_Feeder_e.Init_home_table;
    END_IF

ST115_Feeder_e.Init_home_table:
    IF fb_axis115_10W.xOUT_HOMED THEN
        iCurrentTableIndex := 0;

        IF FEEDER_SIMULATION AND CONST.USE_SIMULATION THEN
            iOUT_Step := ST115_Feeder_e.Init_simu_home_table;
        ELSE
            iOUT_Step := ST115_Feeder_e.Init_table_go_to_zero;
        END_IF
    END_IF

ST115_Feeder_e.Init_simu_home_table:
    IF fb_axis115_10W.xOUT_DONE THEN
        iOUT_Step := ST115_Feeder_e.Init_reset_search_index;
    END_IF

ST115_Feeder_e.Init_table_go_to_zero:
    IF fb_axis115_10W.xOUT_DONE THEN
        iOUT_Step := ST115_Feeder_e.Init_reset_search_index;
    END_IF

ST115_Feeder_e.Init_reset_search_index:
    iSearchIndex := 0;
    fifo.Empty();
    iOUT_Step := ST115_Feeder_e.READY;

ST115_Feeder_e.Init_set_table_pos:
    IF fb_axis115_10W.xOUT_DONE THEN
        iCurrentTableIndex := iCurrentTableIndex + 1;
        iOUT_Step          := ST115_Feeder_e.Init_see_if_piece_there;
    END_IF

ST115_Feeder_e.Init_see_if_piece_there:
    IF simu_feeder.xOUT_NewPiece THEN
        fifo.Put(1);
    END_IF

    IF iSearchIndex < MAX_SEARCH_TURN THEN
        iOUT_Step    := ST115_Feeder_e.Init_set_table_pos;
        iSearchIndex := iSearchIndex + 1;
    ELSE
        iOUT_Step := ST115_Feeder_e.READY;
    END_IF

(***** READY / INIT DONE *****)
ST115_Feeder_e.READY: (* Start AUTO,END,LEER,STEP *)
    IF xIN_Start THEN //IF rtSTART.Q THEN
        iOUT_Step := ST115_Feeder_e.START;
    END_IF

(***** START  ZYKLISCH *****)
ST115_Feeder_e.START: (*  *)
    IF xIN_NextStep AND pxFG_Freigabe^ THEN
        iOUT_Step := ST115_Feeder_e.check_if_feeding_necessary;
    END_IF;

ST115_Feeder_e.check_if_feeding_necessary:
    IF fifo.IsFull() THEN
        iOUT_Step := ST115_Feeder_e.DONE;
    ELSE
        iOUT_Step := ST115_Feeder_e.wait_on_a_piece;
    END_IF

ST115_Feeder_e.wait_on_a_piece:
    IF (FEEDER_SIMULATION AND CONST.USE_SIMULATION AND NOT simu_fifo_feeder_to_rotTable.IsEmpty()) OR
       (NOT (FEEDER_SIMULATION AND CONST.USE_SIMULATION) AND fb_feeder.xIN_PieceInEnd) THEN
        iOUT_Step := ST115_Feeder_e.load_piece;
        simu_fifo_feeder_to_rotTable.Pop(1);
    END_IF

ST115_Feeder_e.load_piece:
    IF NOT fb_axis115_10W.xOUT_DONE THEN
        iOUT_Step := ST115_Feeder_e.wait_rotary_table_done;
    END_IF

ST115_Feeder_e.wait_rotary_table_done:
    IF fb_axis115_10W.xOUT_DONE THEN
        fifo.Put(1);
        iOUT_Step := ST115_Feeder_e.check_if_feeding_necessary;
    END_IF

(***** DONE *****)
ST115_Feeder_e.DONE: (* Letzter Schritt  *)
    IF rtPick.Q THEN
        fifo.Pop(TO_INT(_20_AUTO.recipe.st115.xUseVerLeft));
        fifo.Pop(TO_INT(_20_AUTO.recipe.st115.xUseVerRight));
    END_IF

    IF NOT xIN_AlarmAktiv THEN
        //AUTO
        IF (enIN_State = StateAUTO) AND xIN_RestartCYCL AND NOT fifo.IsFull() THEN
            iOUT_Step := ST115_Feeder_e.START;
            //STEP / END / LEERFAHREN restart
        ELSIF (enIN_State < StateAUTO) AND (enIN_State >= enState.StateSTEP) AND xIN_RestartCYCL AND NOT fifo.IsFull()
            THEN
            iOUT_Step := ST115_Feeder_e.START;
            //STEP / END / LEERFAHREN fertig
        ELSIF (enIN_State = StateREADY) THEN
            iOUT_Step := ST115_Feeder_e.READY;
        END_IF;
    END_IF;

(************ ERROR *************)
ST115_Feeder_e.ERROR: (* ERROR *) ;

END_CASE;

END_FUNCTION_BLOCK

// ---- POUs/20_AUTO/ST120/FB_AUT_120.TcPOU
FUNCTION_BLOCK FB_AUT_120 EXTENDS FB_AUT_ABSTRACT
(****************************************************************************)
(*	POU_AUT_zxx			Bausteinaufrufe Station	zxx							*)
(*	Status				ungetestet											*)
(*  Version:			1.0													*)
(*	Beschrieb:																*)
(*																			*)
(*	Abläufe:			FB_ABLzxxA		Hauptablauf							*)
(*																			*)
(*																			*)
(* 	25.09.2019/Dj															*)
(****************************************************************************)
(*	dd.mm.yyyy   KZ    x.y			Beschrieb								*)
(****************************************************************************)
VAR_INPUT
    (* spezifische Eingänge *)

END_VAR
VAR_OUTPUT
    (* spezifische Ausgänge *)

END_VAR
VAR
    (* Bausteine *)
    fb_Pnp    : FB_ABL_120_Pnp;
    fb_Feeder : FB_ABL_120_Feeder;

    fb_stat_pnp    : FB_AUT_Statistics;
    fb_stat_Feeder : FB_AUT_Statistics;
END_VAR

(*******************************************************************)
(* Timer *)
(*******************************************************************)

(*******************************************************************)
(* Flanken / Merker *)
(*******************************************************************)
//MANU CYCLE
IF (enIN_State = StateMANU) AND xIN_ManuCycle THEN
    xManuCycle := TRUE;
END_IF;

IF (enIN_State <> StateMANU) OR xOUT_Done THEN
    xManuCycle := FALSE;
END_IF

//NEXT STEP
xNextStep := (enIN_State > StateSTEP) OR
             ((enIN_State = StateSTEP) AND xIN_Step) OR
             ((enIN_State = StateMANU) AND xManuCycle);

//RESET
xReset := (enIN_State < StateREADY) AND (enIN_State <> StateINIT) AND NOT xManuCycle;

(*******************************************************************)
(* Bausteinaufrufe Abläufe *)
(*******************************************************************)

xRelease := MAIN.MoverMan.IsProcessUsed(THIS^);

fb_Pnp(xIN_Reset          := xReset,
       xIN_Init           := xIN_Init,
       xIN_Quit           := xIN_Quit,
       xIN_Start          := enIN_State = enState.StateAUTO AND xRelease,
       xIN_Sperre         := NOT xIN_On,
       xIN_NextStep       := xNextStep,
       xIN_AlarmAktiv     := xIN_AlarmAktiv,
       xIN_DryCycle       := xIN_DryCycle,
       xIN_RestartCYCL    := enIN_State >= enState.StateLEER,
       enIN_State         := enIN_State,
       tIN_Timeout        := tIN_Timeout,
       pxFG_Freigabe      := ADR(xRelease),
       Mover              := THIS^.Mover,
       xIN_PceReadyToPick := ST120_Feeder_e.wait_pce_picked = fb_Feeder.iOUT_Step);

fb_Feeder(xIN_Reset          := xReset,
          xIN_Init           := xIN_Init,
          xIN_Quit           := xIN_Quit,
          xIN_Start          := enIN_State >= enState.StateLEER AND xRelease,
          xIN_Sperre         := NOT xIN_On,
          xIN_NextStep       := xNextStep,
          xIN_AlarmAktiv     := xIN_AlarmAktiv,
          xIN_DryCycle       := xIN_DryCycle,
          xIN_RestartCYCL    := enIN_State >= enState.StateLEER,
          enIN_State         := enIN_State,
          tIN_Timeout        := tIN_Timeout,
          pxFG_Freigabe      := ADR(xRelease),
          xIN_PickPiece      := fb_Pnp.xOUT_PickPiece,
          xIN_PnpGripperOpen := TRUE, // TODO replace by sensor of gripper open
          xIN_PnpNotOnTheWay := (ST120_Axis.axis120_02Z.rActPos < 20.0) OR
                                (ST120_Axis.axis120_01Y.rActPos < 100.0));

fb_stat_pnp(xIN_Enable  := enState.StateAUTO = enIN_State,
            xIN_Waiting := fb_Pnp.xOUT_Wait,
            xIN_Running := (fb_Pnp.iOUT_Step >= ST120_Pnp_e.START) AND
                           (fb_Pnp.iOUT_Step <= ST120_Pnp_e.DONE),
            // Since we use a mover system, a cycle is done when we are waiting on a mover
            xIN_Done := fb_Pnp.iOUT_Step = ST120_Pnp_e.waitOnMover);

fb_stat_Feeder(xIN_Enable  := enState.StateAUTO = enIN_State,
               xIN_Waiting := fb_feeder.xOUT_Wait,
               xIN_Running := (fb_feeder.iOUT_Step >= ST120_Feeder_e.START) AND
                              (fb_feeder.iOUT_Step <= ST120_Feeder_e.DONE),
               xIN_Done := fb_feeder.iOUT_Step = ST120_Feeder_e.DONE);

(*******************************************************************)
(* Mover reset flags *)
(*******************************************************************)

(*******************************************************************)
(* OUTPUT *)
(*******************************************************************)
xOUT_InitDone := fb_Pnp.xOUT_InitDone AND fb_Feeder.xOUT_InitDone;
xOUT_Ready    := fb_Pnp.xOUT_Ready AND fb_Feeder.xOUT_Ready;
xOUT_Done     := fb_Pnp.xOUT_Done; // we ignore feeder
xOUT_ErrFlag  := fb_Pnp.xOUT_ErrFlag OR fb_Feeder.xOUT_ErrFlag;
xOUT_Wait     := fb_Pnp.xOUT_Wait OR fb_Feeder.xOUT_Wait;
xOUT_AlarmST  := xOUT_ErrFlag;

IF fb_Pnp.xOUT_ErrFlag THEN
    bOUT_ErrorNum := fb_Pnp.bOUT_Error;
ELSIF fb_Feeder.xOUT_ErrFlag THEN
    bOUT_ErrorNum := fb_Feeder.bOUT_Error;
ELSE
	bOUT_ErrorNum := 0;
END_IF

(*******************************************************************)
(* Bausteinaufruf Error Station *)
(*******************************************************************)
POU_ALARM_120(xIN_QUIT      := xIN_Quit,
              iIN_ArraySize := ST120_Alarm_e._max,
              pstrIN_ALARM  := ADR(HMI.strArALARM[61]),
              refPOU        := THIS^);

(* % of completion of the process *)
PROPERTY iCompletionPC : INT
GET
iCompletionPC := THIS^.fb_Pnp.iOUT_ProcessCompletion;
END_GET
END_PROPERTY

PROPERTY ProcessExecution : ProcessExecution_e
GET
ProcessExecution := THIS^._ProcessExecution;
END_GET
SET
THIS^._ProcessExecution := ProcessExecution;
END_SET
END_PROPERTY

PROPERTY xBusy : BOOL
GET
xBusy := THIS^.fb_Pnp.xOUT_Busy;
END_GET
SET
END_SET
END_PROPERTY

PROPERTY xDone : BOOL
GET
xDone := THIS^.fb_Pnp.xOUT_Ready OR THIS^.fb_Pnp.xOUT_Done;
END_GET
END_PROPERTY

